   VAR
      sUDT_Status { ExternalAccessible := 'False'; ExternalVisible := 'False'; ExternalWritable := 'False'; S7_SetPoint := 'False'} : "UDT_CommonStatus";   // Common status structure
      sR_TRIG_Automatic {InstructionName := 'R_TRIG'; LibVersion := '1.0'; ExternalAccessible := 'False'; ExternalVisible := 'False'; ExternalWritable := 'False'; S7_SetPoint := 'False'} : R_TRIG;   // Rising edge starting automatic mode
      sR_TRIG_PECOn {InstructionName := 'R_TRIG'; LibVersion := '1.0'; ExternalAccessible := 'False'; ExternalVisible := 'False'; ExternalWritable := 'False'; S7_SetPoint := 'False'} : R_TRIG;   // Rising edge trigger PEC on lift conveyor
      sF_TRIG_TIPLiftConveyor {InstructionName := 'F_TRIG'; LibVersion := '1.0'; ExternalAccessible := 'False'; ExternalVisible := 'False'; ExternalWritable := 'False'; S7_SetPoint := 'False'} : F_TRIG;   // Falling edge trigger TIP signal lift conveyor
      sF_TRIG_PECOff {InstructionName := 'F_TRIG'; LibVersion := '1.0'; ExternalAccessible := 'False'; ExternalVisible := 'False'; ExternalWritable := 'False'; S7_SetPoint := 'False'} : F_TRIG;   // Falling edge trigger PEC on lift conveyor
      sx_AutomaticActive { ExternalAccessible := 'False'; ExternalVisible := 'False'; ExternalWritable := 'False'} : Bool;   // Running in automatic
      sx_LoadIsEmptyTote { ExternalAccessible := 'False'; ExternalVisible := 'False'; ExternalWritable := 'False'} : Bool;   // Load on lift conveyor is an empty tote
      sx_LoadIsFullTote { ExternalAccessible := 'False'; ExternalVisible := 'False'; ExternalWritable := 'False'} : Bool;   // Load on lift conveyor is a full tote
      sx_GetEmptyTote { ExternalAccessible := 'False'; ExternalVisible := 'False'; ExternalWritable := 'False'} : Bool;   // Transport empty tote in
      sx_GetFullTote { ExternalAccessible := 'False'; ExternalVisible := 'False'; ExternalWritable := 'False'} : Bool;   // Transport full tote in
      sx_DeliverEmptyTote { ExternalAccessible := 'False'; ExternalVisible := 'False'; ExternalWritable := 'False'} : Bool;   // Transport empty tote out
      sx_DeliverFullTote { ExternalAccessible := 'False'; ExternalVisible := 'False'; ExternalWritable := 'False'} : Bool;   // Transport full tote out
      sx_EmptyRequest { ExternalAccessible := 'False'; ExternalVisible := 'False'; ExternalWritable := 'False'} : Bool;   // Valid empty request active
      sx_FullRequest { ExternalAccessible := 'False'; ExternalVisible := 'False'; ExternalWritable := 'False'} : Bool;   // Valid full request active
      sx_DoEmptyRequest { ExternalAccessible := 'False'; ExternalVisible := 'False'; ExternalWritable := 'False'} : Bool;   // Handle empty request
      sx_DoFullRequest { ExternalAccessible := 'False'; ExternalVisible := 'False'; ExternalWritable := 'False'} : Bool;   // Handle full request
      sx_Idle { ExternalAccessible := 'False'; ExternalVisible := 'False'; ExternalWritable := 'False'} : Bool;   // Transport is Idle
      si_DistanceToOutfeed { ExternalAccessible := 'False'; ExternalVisible := 'False'; ExternalWritable := 'False'} : Int;   // Actual distance to the end of the lift conveyor
      sx_UpperOutfeedingActive { ExternalAccessible := 'False'; ExternalVisible := 'False'; ExternalWritable := 'False'} : Bool;   // Outfeeding to the upper outfeed is on
      sx_LowerOutfeedingActive { ExternalAccessible := 'False'; ExternalVisible := 'False'; ExternalWritable := 'False'} : Bool;   // Outfeeding to the upper outfeed is on
   END_VAR

   VAR CONSTANT
      ci_Up : Int := 2;
      ci_Down : Int := 1;
      ci_DistanceToOutfeed : Int := 39;   // Distance from middle to the end of the lift conveyor
   END_VAR


BEGIN
	(*
	----------------------------------------------------------------------------------------

	Version
	history:
	Date        | Version   | Author        | Remark
	----------------------------------------------------------------------------------------
	07/04/2023  | 3.0       | F.Baten       | First release TIA 17.5
	14/06/2024  | 3.1       | R.Pieczonka   | Changed handshakes connections, added distance counting while outfeeding

	*)


	REGION 1 - Initial
	    REGION 1.1 - Triggers
	        // Starting automatic
	        #sR_TRIG_Automatic(CLK := #iUDT_VSUInterface.Automatic);

	        // Lift conveyor finished TIP
	        #sF_TRIG_TIPLiftConveyor(CLK := #iqUDT_LiftConveyorHandShake.TIP);

	        // Tote arrived on PEC
	        #sF_TRIG_PECOff(CLK := #ix_PECLift);

	        //Tote gone from PEC
	        #sR_TRIG_PECOn(CLK := #ix_PECLift);

	    END_REGION
	END_REGION

	REGION 7 - Automatic mode

	    REGION 7.1 - Determine load on lift
	        // Lift is in upper position and conveyor is ready to send, the empty tote is loaded on the conveyor.
	        IF #ix_SectionIsUp
	            AND #sx_DoEmptyRequest
	            AND #iUDT_LiftConveyorInterface.VFDRunning
	            AND #sF_TRIG_PECOff.Q
	        THEN
	            #sx_LoadIsEmptyTote := TRUE;
	        END_IF;
	        // Lift is in lower position, and outfeeding empty tote.
	        IF #ix_SectionIsDown
	            AND #iUDT_LiftConveyorInterface.VFDRunning
	            AND #sR_TRIG_PECOn.Q
	            AND #sx_LoadIsEmptyTote
	        THEN
	            #sx_LowerOutfeedingActive := TRUE;
	            #si_DistanceToOutfeed := #ci_DistanceToOutfeed;
	        END_IF;

	        IF #sx_LowerOutfeedingActive
	        THEN
	            #si_DistanceToOutfeed -= #iUDT_LiftConveyorInterface.Displacement;
	        END_IF;
	        //If the ditance from middle conveyor to the end of it is reached,  then the information about tote on the lift is cleared.
	        IF #sx_LowerOutfeedingActive
	            AND #si_DistanceToOutfeed <= 0
	        THEN
	            #sx_LowerOutfeedingActive := FALSE;
	            #sx_LoadIsEmptyTote := FALSE;
	        END_IF;

	        // Lift is in lower position and conveyor is ready to send, the full tote is loaded on the conveyor.
	        IF #ix_SectionIsDown
	            AND #sx_DoFullRequest
	            AND #iUDT_LiftConveyorInterface.VFDRunning
	            AND #sF_TRIG_PECOff.Q
	        THEN
	            #sx_LoadIsFullTote := TRUE;
	        END_IF;
	        // Lift is in upper position, and outfeeding full tote.
	        IF #ix_SectionIsUp
	            AND #iUDT_LiftConveyorInterface.VFDRunning
	            AND #sR_TRIG_PECOn.Q
	            AND #sx_LoadIsFullTote
	        THEN
	            #sx_UpperOutfeedingActive := TRUE;
	            #si_DistanceToOutfeed := #ci_DistanceToOutfeed;
	        END_IF;

	        IF #sx_UpperOutfeedingActive
	        THEN
	            #si_DistanceToOutfeed += #iUDT_LiftConveyorInterface.Displacement;
	        END_IF;
	        //If the ditance from middle conveyor to the end of it is reached, then the information about tote on the lift is cleared.
	        IF #sx_UpperOutfeedingActive
	            AND #si_DistanceToOutfeed <= 0
	        THEN
	            #sx_LoadIsFullTote := FALSE;
	            #sx_UpperOutfeedingActive := FALSE;
	        END_IF;

	        // When starting automatic mode and no load is active but pec still occupied, the load will be set as Full tote.
	        IF NOT #sx_LoadIsFullTote
	            AND NOT #sx_LoadIsEmptyTote
	            AND NOT #ix_PECLift
	            AND #sR_TRIG_Automatic.Q
	        THEN
	            #sx_LoadIsFullTote := TRUE;
	        END_IF;

	        IF #sR_TRIG_Automatic.Q
	        THEN
	            #sx_LowerOutfeedingActive := FALSE;
	            #sx_UpperOutfeedingActive := FALSE;
	        END_IF;
	    END_REGION

	    REGION 7.2 - Request totes
	        // request for empty totes : infeed is full and outfeed is empty and both are automatic active
	        #sx_EmptyRequest := #iqUDT_InfeedEmptyUpHandShake.RTS
	        AND #iqUDT_OutfeedEmptyDownHandShake.RTR
	        AND #ix_ConveyorEmptyInAuto
	        AND #ix_ConveyorEmptyOutAuto;

	        // request for full totes : infeed is full and outfeed is empty and both are automatic active
	        #sx_FullRequest := #iqUDT_InfeedFullDownHandShake.RTS
	        AND #iqUDT_OutfeedFullUpHandshakeUpstream.RTR
	        AND #ix_ConveyorFullInAuto
	        AND #ix_ConveyorFullOutAuto;
	    END_REGION

	    REGION 7.3 - Handle request
	        // Setting reqest to be handled
	        IF #sx_EmptyRequest
	            AND NOT #sx_DoFullRequest
	            AND NOT #sx_LoadIsEmptyTote
	        THEN
	            #sx_DoEmptyRequest := TRUE;
	        ELSIF #sx_FullRequest
	            AND NOT #sx_DoEmptyRequest
	            AND NOT #sx_LoadIsFullTote
	        THEN
	            #sx_DoFullRequest := TRUE;
	        END_IF;

	        // Empty tote is loaded
	        IF (#sx_DoEmptyRequest AND #sx_LoadIsEmptyTote)
	        THEN
	            #sx_DoEmptyRequest := FALSE;
	        END_IF;

	        // Full tote is loaded
	        IF (#sx_DoFullRequest AND #sx_LoadIsFullTote)
	        THEN
	            #sx_DoFullRequest := FALSE;
	        END_IF;

	        // Active request is not valid anymore as lift moved to position
	        IF #sx_DoEmptyRequest AND NOT #sx_EmptyRequest AND #iqUDT_InfeedEmptyUpHandShake.RTS AND #ix_SectionIsUp AND #sx_GetEmptyTote THEN
	            #sx_GetEmptyTote := FALSE;
	            #sx_DoEmptyRequest := FALSE;
	        END_IF;

	        IF #sx_DoFullRequest AND NOT #sx_FullRequest AND #iqUDT_InfeedFullDownHandShake.RTS AND #ix_SectionIsDown AND #sx_GetFullTote THEN
	            #sx_GetFullTote := FALSE;
	            #sx_DoFullRequest := FALSE;
	        END_IF;

	    END_REGION

	    REGION 7.4 - Active Transports
	        // Load empty tote transport is active
	        IF #sx_DoEmptyRequest AND #ix_SectionIsUp
	        THEN
	            #sx_GetEmptyTote := TRUE;
	        END_IF;

	        IF #sx_GetEmptyTote
	            AND
	            ((#iUDT_LiftConveyorInterface.ActualSpeed = 0) AND #sx_LoadIsEmptyTote)
	        THEN
	            #sx_GetEmptyTote := FALSE;
	        END_IF;

	        // Load full tote transport is active
	        IF #sx_DoFullRequest AND #ix_SectionIsDown
	        THEN
	            #sx_GetFullTote := TRUE;
	        END_IF;

	        IF #sx_GetFullTote AND #sx_LoadIsFullTote AND (#iUDT_LiftConveyorInterface.ActualSpeed = 0)
	        THEN
	            #sx_GetFullTote := FALSE;
	        END_IF;

	        // Deliver transports are active
	        #sx_DeliverEmptyTote := #ix_SectionIsDown AND #sx_LoadIsEmptyTote AND (#iUDT_LiftConveyorInterface.ActualSpeed <> 0);
	        #sx_DeliverFullTote := #ix_SectionIsUp AND #sx_LoadIsFullTote AND (#iUDT_LiftConveyorInterface.ActualSpeed <> 0);

	        // Transport is idle
	        #sx_Idle := NOT #sx_GetEmptyTote
	        AND NOT #sx_GetFullTote
	        AND NOT #sx_DeliverFullTote
	        AND NOT #sx_DeliverEmptyTote;
	    END_REGION

	    REGION 7.5 - Lift position request
	        // When lift is at level and transports finished (free to move)
	        // To go to lower level (bring empty tote or get full one)
	        IF #sx_Idle
	            AND ((#ix_SectionIsUp AND #sx_DoFullRequest)
	            OR #sx_LoadIsEmptyTote)
	        THEN
	            #qi_RequestedPosition := #ci_Down;
	        END_IF;

	        // To go to upper level (bring full tote or get empty one)
	        IF #sx_Idle
	            AND ((#ix_SectionIsDown AND #sx_DoEmptyRequest) OR #sx_LoadIsFullTote)
	        THEN
	            #qi_RequestedPosition := #ci_Up;
	        END_IF;

	        #qx_TransportIdle := #sx_Idle;

	    END_REGION

	END_REGION

	REGION 8 - Handshake to conveyors
	    // Reset when not connected
	    #iqUDT_InfeedEmptyUpHandShake.RTR := FALSE;
	    #iqUDT_InfeedFullDownHandShake.RTR := FALSE;

	    #iqUDT_LiftConveyorHandShakeUpstream.GIN := 0;
	    #iqUDT_LiftConveyorHandShakeUpstream.NrOfPosToShift := 0;
	    #iqUDT_OutfeedFullUpHandShake.GIN := 0;
	    #iqUDT_OutfeedFullUpHandShake.NrOfPosToShift := 0;
	    #iqUDT_OutfeedEmptyDownHandShake.GIN := 0;
	    #iqUDT_OutfeedEmptyDownHandShake.NrOfPosToShift := 0;

	    // Direct interface signals when on level
	    IF #ix_SectionIsUp THEN
	        #qx_LiftConveyorDirection := TRUE;                  // Changing direction to left
	        // Infeed
	        #iqUDT_InfeedEmptyUpHandShake.RTR := #iqUDT_LiftConveyorHandShake.RTR AND (#sx_EmptyRequest OR #iqUDT_InfeedEmptyUpHandShake.TIP);
	        #iqUDT_LiftConveyorHandShake.GIN := #iqUDT_InfeedEmptyUpHandShake.GIN;
	        #iqUDT_LiftConveyorHandShakeUpstream.NrOfPosToShift := #iqUDT_InfeedEmptyUpHandShake.NrOfPosToShift;
	        #iqUDT_InfeedEmptyUpHandShake.NrOfPosToShift := 0;
	        #iqUDT_LiftConveyorHandShakeUpstream.RTS := #iqUDT_InfeedEmptyUpHandShake.RTS;
	        //  #iqUDT_HandShakeLiftUp.TIP := #iqUDT_HandShakeEmptyIn.TIP;
	        #iqUDT_LiftConveyorHandShakeUpstream.ResetEnergySave := #iqUDT_InfeedEmptyUpHandShake.ResetEnergySave;

	        // Outfeed
	        #iqUDT_OutfeedFullUpHandshakeUpstream.RTS := #iqUDT_LiftConveyorHandShake.RTS AND #sx_LoadIsFullTote;
	        #iqUDT_OutfeedFullUpHandshakeUpstream.TIP := #iqUDT_LiftConveyorHandShake.TIP;
	        #iqUDT_OutfeedFullUpHandshakeUpstream.GIN := #iqUDT_LiftConveyorHandShake.GIN;
	        #iqUDT_OutfeedFullUpHandshakeUpstream.NrOfPosToShift := #iqUDT_LiftConveyorHandShake.NrOfPosToShift;
	        #iqUDT_LiftConveyorHandShake.NrOfPosToShift := 0;

	        // lift to outfeed transport
	        #iqUDT_LiftConveyorHandShakeUpstream.RTR := #iqUDT_OutfeedFullUpHandshakeUpstream.RTR AND (#sx_LoadIsFullTote OR #iqUDT_LiftConveyorHandShake.TIP);
	    END_IF;

	    IF #ix_SectionIsDown THEN
	        #qx_LiftConveyorDirection := FALSE;                 //Changing direction to right

	        // Infeed Full to lift
	        #iqUDT_InfeedFullDownHandShake.RTR := #iqUDT_LiftConveyorHandShakeUpstream.RTR AND (#sx_FullRequest OR #iqUDT_InfeedFullDownHandShake.TIP);
	        #iqUDT_LiftConveyorHandShakeUpstream.GIN := #iqUDT_InfeedFullDownHandShake.GIN;
	        #iqUDT_LiftConveyorHandShakeUpstream.NrOfPosToShift := #iqUDT_InfeedFullDownHandShake.NrOfPosToShift;
	        #iqUDT_InfeedFullDownHandShake.NrOfPosToShift := 0;
	        #iqUDT_LiftConveyorHandShakeUpstream.RTS := #iqUDT_InfeedFullDownHandShake.RTS;
	        #iqUDT_LiftConveyorHandShakeUpstream.TIP := #iqUDT_InfeedFullDownHandShake.TIP;
	        #iqUDT_LiftConveyorHandShakeUpstream.ResetEnergySave := #iqUDT_InfeedFullDownHandShake.ResetEnergySave;

	        // Outfeed
	        #iqUDT_OutfeedEmptyDownHandshakeUpstream.RTS := #iqUDT_LiftConveyorHandShakeUpstream.RTS AND #sx_LoadIsEmptyTote;
	        #iqUDT_OutfeedEmptyDownHandshakeUpstream.TIP := #iqUDT_LiftConveyorHandShake.TIP;
	        #iqUDT_OutfeedEmptyDownHandshakeUpstream.GIN := #iqUDT_LiftConveyorHandShake.GIN;
	        #iqUDT_OutfeedEmptyDownHandshakeUpstream.NrOfPosToShift := #iqUDT_LiftConveyorHandShake.NrOfPosToShift;
	        #iqUDT_LiftConveyorHandShake.NrOfPosToShift := 0;

	        // lift to outfeed transport
	        #iqUDT_LiftConveyorHandShake.RTR := #iqUDT_OutfeedEmptyDownHandshakeUpstream.RTR AND (#sx_LoadIsEmptyTote OR #iqUDT_LiftConveyorHandShake.TIP);

	    END_IF;

	    #iqUDT_OutfeedFullUpHandshakeUpstream.ResetEnergySave := #iqUDT_InfeedFullDownHandShake.ResetEnergySave
	    OR #iqUDT_LiftConveyorHandShake.ResetEnergySave
	    AND #ix_SectionIsUp;
	    #iqUDT_OutfeedEmptyDownHandshakeUpstream.ResetEnergySave := #iqUDT_InfeedEmptyUpHandShake.ResetEnergySave
	    OR #iqUDT_LiftConveyorHandShake.ResetEnergySave
	    AND #ix_SectionIsDown;

	    //Stop when NOT on level
	    #qx_HoldLiftConveyor := NOT #ix_SectionIsDown AND NOT #ix_SectionIsUp;

	END_REGION

END_FUNCTION_BLOCK

FUNCTION_BLOCK "FB_PECUpdate"
TITLE = FB_PECUpdate
{ S7_Optimized_Access := 'TRUE' }
AUTHOR : MHSE
FAMILY : GeneralSystemFunctions
VERSION : 3.0
// ATTRIBUTES
// AUTO_NUMBER = True
// BLOCK_NUMBER = 221
// END_ATTRIBUTES
//Function block to update parcel data in a tracking array at PEC position.
   VAR_INPUT
      iUDT_PECUpdateConfiguration { ExternalAccessible := 'False'; ExternalVisible := 'False'; ExternalWritable := 'False'} : "UDT_PECUpdateConfiguration";   //   PEC update configuration
      iUDT_ConveyorCommonConfiguration { ExternalAccessible := 'False'; ExternalVisible := 'False'; ExternalWritable := 'False'} : "UDT_ConveyorCommonConfiguration";   //   Conveyor configuration
      ix_PEC { ExternalAccessible := 'False'; ExternalVisible := 'False'; ExternalWritable := 'False'} : Bool;   //   TRUE when the end of section photoeye is not blocked
      ix_TeachingMode { ExternalAccessible := 'False'; ExternalVisible := 'False'; ExternalWritable := 'False'} : Bool;   //   Teaching mode enable
   END_VAR

   VAR_OUTPUT
      qUDT_Status { ExternalAccessible := 'False'; ExternalVisible := 'False'; ExternalWritable := 'False'} : "UDT_PECUpdateStatus";   //   Status structure
      qi_GINwrite { ExternalAccessible := 'False'; ExternalVisible := 'False'; ExternalWritable := 'False'} : Int;   //  Gin found or generated
      qx_PECFiltered { ExternalAccessible := 'False'; ExternalVisible := 'False'; ExternalWritable := 'False'} : Bool;   //   Filtered photoeye signal
   END_VAR

   VAR_IN_OUT
      iqUDT_ConveyorInterface : "UDT_ConveyorInterface";   //   Conveyor interface
      iqUDT_UnknownGINRange : "UDT_UnknownGIN";   //   Unknown GIN
      iqUDT_FifoHeader : "UDT_FifoHeader";   //   FIFO header
      iqUDT_Statistics : "UDT_PECUpdateStatistics";   //   Statistic structure
      iqa_TrackingData : Array[*] of Int;   //   Tracking data
      iqa_FifoData : Array[*] of Int;   //   FIFO data
   END_VAR

   VAR
      sFB_PEC { ExternalAccessible := 'False'; ExternalVisible := 'False'; ExternalWritable := 'False'; S7_SetPoint := 'False'} : "FB_PEC";   //   Photoeye function
      sFB_LengthMeasurement { ExternalAccessible := 'False'; ExternalVisible := 'False'; ExternalWritable := 'False'; S7_SetPoint := 'False'} : "FB_ParcelLength";   //   Length measurement
      sUDT_LostGINFIFOStatus { ExternalAccessible := 'False'; ExternalVisible := 'False'; ExternalWritable := 'False'; S7_SetPoint := 'False'} : "UDT_FifoStatus";   //   Lost GIN FIFO status
      ss_PECDataDeviation { ExternalAccessible := 'False'; ExternalVisible := 'False'; ExternalWritable := 'False'} : Struct   // PEC/Data deviation calculation structure
         Last { ExternalAccessible := 'False'; ExternalVisible := 'False'; ExternalWritable := 'False'} : Int;   //  Last deviation [cm]
         GIN { ExternalAccessible := 'False'; ExternalVisible := 'False'; ExternalWritable := 'False'} : Int;   //  Last GIN deviation
         Sum { ExternalAccessible := 'False'; ExternalVisible := 'False'; ExternalWritable := 'False'} : Int;   //  Deviation sum [cm]
         Nr { ExternalAccessible := 'False'; ExternalVisible := 'False'; ExternalWritable := 'False'} : Int;   //  Deviation number
      END_STRUCT;
      ss_ValidGINRange { ExternalAccessible := 'False'; ExternalVisible := 'False'; ExternalWritable := 'False'} : Struct   //   Valid GIN range
         Start { ExternalAccessible := 'False'; ExternalVisible := 'False'; ExternalWritable := 'False'} : Int;
         End { ExternalAccessible := 'False'; ExternalVisible := 'False'; ExternalWritable := 'False'} : Int;
         GIN { ExternalAccessible := 'False'; ExternalVisible := 'False'; ExternalWritable := 'False'} : Int;
      END_STRUCT;
      ss_AlignedParcelsCounters { ExternalAccessible := 'False'; ExternalVisible := 'False'; ExternalWritable := 'False'} : Struct   //   Aligned parcels counters
         Total { ExternalAccessible := 'False'; ExternalVisible := 'False'; ExternalWritable := 'False'} : Int;   //   Total aligned parcels
         DataNoPEC { ExternalAccessible := 'False'; ExternalVisible := 'False'; ExternalWritable := 'False'} : Int;   //   Parcels aligned in case data detected without photoeye signal
         PECNoData { ExternalAccessible := 'False'; ExternalVisible := 'False'; ExternalWritable := 'False'} : Int;   //   Parcels aligned in case parcel detected without data
      END_STRUCT;
      ss_LostParcelsCounters { ExternalAccessible := 'False'; ExternalVisible := 'False'; ExternalWritable := 'False'} : Struct   //   Lost parcels counters
         Total { ExternalAccessible := 'False'; ExternalVisible := 'False'; ExternalWritable := 'False'} : Int;   //   Total number of lost parcels
         DoubleData { ExternalAccessible := 'False'; ExternalVisible := 'False'; ExternalWritable := 'False'} : Int;   //   Parcels lost due to double data found in a search window
         ParcelNotFound { ExternalAccessible := 'False'; ExternalVisible := 'False'; ExternalWritable := 'False'} : Int;   //   Parcels lost due to no parcel detected after travelling search window distance
      END_STRUCT;
      ss_LostValidParcelsCounters { ExternalAccessible := 'False'; ExternalVisible := 'False'; ExternalWritable := 'False'} : Struct   //   Lost parcels counters
         Total { ExternalAccessible := 'False'; ExternalVisible := 'False'; ExternalWritable := 'False'} : Int;   //   Total number of lost parcels
         DoubleData { ExternalAccessible := 'False'; ExternalVisible := 'False'; ExternalWritable := 'False'} : Int;   //   Parcels lost due to double data found in a search window
         ParcelNotFound { ExternalAccessible := 'False'; ExternalVisible := 'False'; ExternalWritable := 'False'} : Int;   //   Parcels lost due to no parcel detected after travelling search window distance
      END_STRUCT;
      si_UnknownParcelsCounters { ExternalAccessible := 'False'; ExternalVisible := 'False'; ExternalWritable := 'False'} : Struct   //   Unknown parcels counters
         Total { ExternalAccessible := 'False'; ExternalVisible := 'False'; ExternalWritable := 'False'} : Int;   //   Total number of unknown parcels
         LostParcelFound { ExternalAccessible := 'False'; ExternalVisible := 'False'; ExternalWritable := 'False'} : Int;   //   Parcel found with a lost data, unknown GIN created
         DataNotFound { ExternalAccessible := 'False'; ExternalVisible := 'False'; ExternalWritable := 'False'} : Int;   //   Data not found during search window scan
      END_STRUCT;
      sR_TRIG_Parcel {InstructionName := 'R_TRIG'; LibVersion := '1.0'; ExternalAccessible := 'False'; ExternalVisible := 'False'; ExternalWritable := 'False'; S7_SetPoint := 'False'} : R_TRIG;   //   Parcel detected rising edge to count parcels
      sR_TRIG_ParcelFound {InstructionName := 'R_TRIG'; LibVersion := '1.0'; ExternalAccessible := 'False'; ExternalVisible := 'False'; ExternalWritable := 'False'; S7_SetPoint := 'False'} : R_TRIG;   //   Parcel detected rising edge to update the PEC position tracking record
      sR_TRIG_DataFound {InstructionName := 'R_TRIG'; LibVersion := '1.0'; ExternalAccessible := 'False'; ExternalVisible := 'False'; ExternalWritable := 'False'; S7_SetPoint := 'False'} : R_TRIG;   //   Any data found at a PEC position rising edge
      sR_TRIG_PositiveDataFound {InstructionName := 'R_TRIG'; LibVersion := '1.0'; ExternalAccessible := 'False'; ExternalVisible := 'False'; ExternalWritable := 'False'; S7_SetPoint := 'False'} : R_TRIG;   //   Positive data found at a PEC position rising edge
      sR_TRIG_TeachMode {InstructionName := 'R_TRIG'; LibVersion := '1.0'; ExternalAccessible := 'False'; ExternalVisible := 'False'; ExternalWritable := 'False'; S7_SetPoint := 'False'} : R_TRIG;   //   Teaching mode activation rising edge
      sR_TRIG_TooManyLost {InstructionName := 'R_TRIG'; LibVersion := '1.0'; ExternalAccessible := 'False'; ExternalVisible := 'False'; ExternalWritable := 'False'; S7_SetPoint := 'False'} : R_TRIG;   //   Too many lost parcels error statistics trigger
      slr_Performance { ExternalAccessible := 'False'; ExternalVisible := 'False'; ExternalWritable := 'False'} : LReal := 100.0;   //   Update performance [%]
      sdi_TotalNumberOfParcels { ExternalAccessible := 'False'; ExternalVisible := 'False'; ExternalWritable := 'False'} : DInt;   //   Total number of parcels detected
      sdi_TotalNumberOfData { ExternalAccessible := 'False'; ExternalVisible := 'False'; ExternalWritable := 'False'} : DInt;   //   Total number of data detected
      si_PECPosition { ExternalAccessible := 'False'; ExternalVisible := 'False'; ExternalWritable := 'False'} : Int;   //   Photoeye position [cm]
      si_SearchWindow { ExternalAccessible := 'False'; ExternalVisible := 'False'; ExternalWritable := 'False'} : Int;   //   Data search distance from photoeye position [cm]
      si_GINToWrite { ExternalAccessible := 'False'; ExternalVisible := 'False'; ExternalWritable := 'False'} : Int;   //   Found or generated GIN, which will be used to update photoeye position in the tracking array
      si_PositionToUpdate { ExternalAccessible := 'False'; ExternalVisible := 'False'; ExternalWritable := 'False'} : Int;   //   Position in a tracking array to be updated
      si_Direction { ExternalAccessible := 'False'; ExternalVisible := 'False'; ExternalWritable := 'False'} : Int;   //   Direction of the displacement to parametrize loops
      si_Displacement { ExternalAccessible := 'False'; ExternalVisible := 'False'; ExternalWritable := 'False'} : Int;   //   Displacement [cm]
      si_ParcelWaitDistance { ExternalAccessible := 'False'; ExternalVisible := 'False'; ExternalWritable := 'False'} : Int;   //   Parcel delay [cm]
      si_LastUpdatedGIN { ExternalAccessible := 'False'; ExternalVisible := 'False'; ExternalWritable := 'False'} : Int;   //   Last updated GIN to check if next data is a new one
      si_LastCountedData { ExternalAccessible := 'False'; ExternalVisible := 'False'; ExternalWritable := 'False'} : Int;   //   Last counted data
      si_LostParcelsInARow { ExternalAccessible := 'False'; ExternalVisible := 'False'; ExternalWritable := 'False'} : Int;   //   Number of lost parcel in a row
      si_NumberOfTeachedParcels { ExternalAccessible := 'False'; ExternalVisible := 'False'; ExternalWritable := 'False'} : Int;   //   Number of teached parcels
      si_AverageSlip { ExternalAccessible := 'False'; ExternalVisible := 'False'; ExternalWritable := 'False'} : Int;   //   Average parcel slip [cm]
      si_CalculatedLengthCorrection { ExternalAccessible := 'False'; ExternalVisible := 'False'; ExternalWritable := 'False'} : Int;   //   Calculated length correction after teaching
      si_ParcelLengthFilterCounter { ExternalAccessible := 'False'; ExternalVisible := 'False'; ExternalWritable := 'False'} : Int;   //  Parcel length filter counter [cm]
      si_ParcelLengthFilterOldGIN { ExternalAccessible := 'False'; ExternalVisible := 'False'; ExternalWritable := 'False'} : Int;   //  Parcel length filter old GIN
      si_LoopCounter { ExternalAccessible := 'False'; ExternalVisible := 'False'; ExternalWritable := 'False'} : Int;   //   Loop counter
      sx_ParcelDetected { ExternalAccessible := 'False'; ExternalVisible := 'False'; ExternalWritable := 'False'} : Bool;   //   Parcel detected
      sx_ParcelWaitEnable { ExternalAccessible := 'False'; ExternalVisible := 'False'; ExternalWritable := 'False'} : Bool;   //   Missing parcel monitoring
      sx_TeachingMode { ExternalAccessible := 'False'; ExternalVisible := 'False'; ExternalWritable := 'False'} : Bool;   //   Teaching mode
      sx_GenerateGIN { ExternalAccessible := 'False'; ExternalVisible := 'False'; ExternalWritable := 'False'} : Bool;   //   Request to generate GIN
      sx_LostGINFIFOError { ExternalAccessible := 'False'; ExternalVisible := 'False'; ExternalWritable := 'False'} : Bool;   //   Lost GIN FIFO error
      sx_LostGINFIFOWarning { ExternalAccessible := 'False'; ExternalVisible := 'False'; ExternalWritable := 'False'} : Bool;   //   Lost GIN FIFO warning
      sx_InvalidDirection { ExternalAccessible := 'False'; ExternalVisible := 'False'; ExternalWritable := 'False'} : Bool;   //   Invalid direction
      sx_InvalidGINRange { ExternalAccessible := 'False'; ExternalVisible := 'False'; ExternalWritable := 'False'} : Bool;   //   Invalid GIN range
      sx_InvalidDisplacement { ExternalAccessible := 'False'; ExternalVisible := 'False'; ExternalWritable := 'False'} : Bool;   //   Invalid displacement
      sx_InvalidSearchWindow { ExternalAccessible := 'False'; ExternalVisible := 'False'; ExternalWritable := 'False'} : Bool;   //   Invalid search window
      sx_DoubleDataFound { ExternalAccessible := 'False'; ExternalVisible := 'False'; ExternalWritable := 'False'} : Bool;   //   Double data detected
      sx_LengthMeasurementEnable { ExternalAccessible := 'False'; ExternalVisible := 'False'; ExternalWritable := 'False'} : Bool;
   END_VAR

   VAR_TEMP
      tUDT_PECConfiguration : "UDT_PECConfiguration";   //   PEC configuration
      tUDT_PECStatus : "UDT_PECStatus";   //   PEC status
   END_VAR

   VAR CONSTANT
      ci_ZeroGIN : Int;   //   GIN = 0
   END_VAR


BEGIN
	(*
	----------------------------------------------------------------------------------------

	Version history:
	Date        | Version   | Author        | Remark
	----------------------------------------------------------------------------------------
	24/05/2019  | 0.1       | L.Klar        | first release MHSE TIA 15.1
	13/06/2019  | 0.2       | A.Nowak       | Replacement of instruction if for direct write into variable
	21/06/2019  | 0.3       | A.Nowak       | Add gap mesurement function and reorganise block (regions)
	24/07/2019  | 2.0       | L.Klar        | 2.0 MHSE library release TIA 15.1
	23/08/2019  | 2.1       | L.Klar        | "UDT_ConveyorConfiguration" changed to "UDT_ConveyorCommonConfiguration"
	XX/08/2019  | 2.2       | L.Klar        | Update logic changed
	19/09/2019  | 2.3       | P.Majka       | Updating checking PEC and PEC filtered signals
	30/09/2019  | 2.4       | L.Klar        | FB_PEC added, Filtered PEC signal output added
	21/10/2019  | 2.6       | L.Klar        | Configuration UDT chanaged to input, PEC configuration interface input name changed
	23/10/2019  | 2.7       | P.Majka       | Added Region 1, renumerating Regions, changed logic in Region 10.3 and Region 5
	29/10/2019  | 2.8       | L.Klar        | FB_PEC call changed
	14/11/2019  | 2.9       | L.Klar        | Deviations calculation corrected
	14/11/2019  | 3.0       | P.Majka       | 3.0 MHSE library release TIA 15.1
	20/12/2019  | 3.1       | S.Deulkar     | Used configureation error bit to report to conveyor block
	07/01/2020  | 3.2       | L.Klar        | GIN record structure updated, GIN cleared with default one during generation
	                                        | PECUpdate configuration UDT update - search window DINT -> INT,
	                                        | Conveyor common configuration UDT update - length INT -> DINT  conversion added
	29/01/2020  | 3.3       | L.Klar        | Negative GIN handling fixed, configuration bit added to delete negative GIN instead of ignoing it.
	24/02/2020  | 3.4       | L.Klar        | Formating changes, statistics counter added
	10/03/2020  | 3.5       | F.Baten       | Range check unknown GIN region 7
	26/03/2020  | 3.6       | F.Baten       | Added output 'qi_GINwrite'
	25/11/2020  | 3.7       | L.Klar        | Length filter added
	07/12/2020  | 3.8       | L.Klar        | Length filter bug fix
	22/01/2021  | 3.9       | L.Klar        | Total number of parcels and lost parcels counter fixed
	14/08/2021  | 3.10      | S. Deulkar    | Update from EMA
	21/02/2023  | 4.0       | F.Baten       | 4.0 Release TIA 17.5
	*)


	REGION 1 – FIFO header status update

	    "FC_Fifo"(ic_Mode := 'S',
	              qUDT_Status => #sUDT_LostGINFIFOStatus,
	              qx_Error => #sx_LostGINFIFOError,
	              qx_Warning => #sx_LostGINFIFOWarning,
	              iqv_Data := #si_GINToWrite,
	              iqUDT_FifoHeader := #iqUDT_FifoHeader,
	              iqv_DataBuffer := #iqa_FifoData);

	END_REGION

	REGION 2 – Displacement read

	    #si_Displacement := #iqUDT_ConveyorInterface.Displacement;

	END_REGION

	REGION 3 – PEC Position conversion from mm to cm

	    // The conversion is required because the photoeye position is given in mm and the tracking resolution is 1 cm.
	    #si_PECPosition := DINT_TO_INT(#iUDT_PECUpdateConfiguration.Distance / 10);

	END_REGION

	REGION 4 – Teaching mode enable

	    (* Teaching mode is used to calculate conveyor length correction, which allows to align real conveyor length with a tracking array length.
	       Correction is calculated as a difference between photoeye signal and tracking data deviations.
	       Calculated correction has to be manually copied from a FB_PECUpdate instance data block to conveyor configuration.*)

	    // Teaching mode is initialized and activated manually via block input.
	    #sR_TRIG_TeachMode(CLK := #ix_TeachingMode);

	    IF (#sR_TRIG_TeachMode.Q
	        AND NOT #sx_TeachingMode)
	    THEN
	        #ss_PECDataDeviation.Nr := 0;
	        #ss_PECDataDeviation.Sum := 0;
	        #si_NumberOfTeachedParcels := 0;
	        #sx_TeachingMode := TRUE;
	    END_IF;

	END_REGION

	REGION 5 – Photoeye

	    (*FB_PEC block call to filter photoeye signal and calculate jam status.*)

	    // Copy PEC configuration.
	    #tUDT_PECConfiguration.Distance := #iUDT_PECUpdateConfiguration.Distance;
	    #tUDT_PECConfiguration.JamDisplacementLimit := #iUDT_PECUpdateConfiguration.JamDisplacementLimit;
	    #tUDT_PECConfiguration.TimeOnDelay := #iUDT_PECUpdateConfiguration.TimeOnDelay;
	    #tUDT_PECConfiguration.TimeOffDelay := #iUDT_PECUpdateConfiguration.TimeOffDelay;
	    #tUDT_PECConfiguration.ResetWithPECBlocked := #iUDT_PECUpdateConfiguration.ResetWithPECBlocked;

	    //Call FB_PEC.
	    #sFB_PEC(ix_PEC := #ix_PEC,
	             iUDT_PECConfiguration := #tUDT_PECConfiguration,
	             qUDT_HMIStatus => #tUDT_PECStatus,
	             iqUDT_ConveyorInterface := #iqUDT_ConveyorInterface,
	             iqUDT_PECStatistics := #iqUDT_Statistics.PEC);

	    // Parcel length filter
	    IF NOT #ix_PEC
	        AND #iUDT_PECUpdateConfiguration.ParcelLengthFilter
	        AND #iqa_TrackingData[#si_PECPosition - 1] > 0
	        AND #iqa_TrackingData[#si_PECPosition - 1] <> #si_ParcelLengthFilterOldGIN THEN

	        IF "DB_GIN".GIN[#iqa_TrackingData[#si_PECPosition - 1]].General.Length > 0 THEN
	            #si_ParcelLengthFilterCounter := "DB_GIN".GIN[#iqa_TrackingData[#si_PECPosition - 1]].General.Length;
	        END_IF;

	        #si_ParcelLengthFilterOldGIN := #iqa_TrackingData[#si_PECPosition - 1];

	    END_IF;

	    IF #si_ParcelLengthFilterCounter > 0 THEN

	        #qUDT_Status.PEC := FALSE;
	        #qx_PECFiltered := FALSE;
	        #si_ParcelLengthFilterCounter -= #iqUDT_ConveyorInterface.Displacement;

	    ELSE

	        #qUDT_Status.PEC := #sFB_PEC.qx_PECFiltered;
	        #qx_PECFiltered := #sFB_PEC.qx_PECFiltered;

	    END_IF;

	    #qUDT_Status.Jam := #tUDT_PECStatus.Jam;

	    // Parcel detected variable to simplify further photoeye position tracking record update.
	    #sx_ParcelDetected := NOT #qUDT_Status.PEC;

	END_REGION

	REGION 6 – Error reset

	    // Reset errors when reset signal is given.
	    IF (#iqUDT_ConveyorInterface.InternalErrorReset)
	    THEN
	        #si_LostParcelsInARow := 0;
	        #qUDT_Status.TooManyLost := FALSE;
	        #sx_InvalidDisplacement := FALSE;
	    END_IF;

	END_REGION

	REGION 7 – GIN generator initialization

	    // Valid GIN range configuration is moved to a structure.
	    #ss_ValidGINRange.Start := #iUDT_PECUpdateConfiguration.GINRangeStart;
	    #ss_ValidGINRange.End := #iUDT_PECUpdateConfiguration.GINRangeEnd;

	    // Check if the unknown GIN is within range
	    IF #iqUDT_UnknownGINRange.GIN < #iqUDT_UnknownGINRange.Start
	        OR #iqUDT_UnknownGINRange.GIN > #iqUDT_UnknownGINRange.End
	    THEN
	        #iqUDT_UnknownGINRange.GIN := #iqUDT_UnknownGINRange.Start;
	    END_IF;

	    // Whenever valid GIN range is changed and the generated GIN doesn't fit, it's initialized.
	    IF (#ss_ValidGINRange.GIN < #ss_ValidGINRange.Start
	        OR #ss_ValidGINRange.GIN > #ss_ValidGINRange.End)
	    THEN
	        #ss_ValidGINRange.GIN := #ss_ValidGINRange.Start;
	    END_IF;

	    // Valid GIN range is set locally in PEC update configuration structure and it can't overlap with a global unknown GIN range.
	    #sx_InvalidGINRange := #iUDT_PECUpdateConfiguration.GenerationPoint
	    AND (#ss_ValidGINRange.End <= #ss_ValidGINRange.Start
	    OR #ss_ValidGINRange.Start <= #iqUDT_UnknownGINRange.End
	    OR #iqUDT_UnknownGINRange.End <= #iqUDT_UnknownGINRange.Start)
	    AND #ss_ValidGINRange.Start < 1000;   // Until 1000 it is UFO range

	END_REGION

	REGION 8 – Search window and displacement validation

	    (*Both parameters have to be checked to prevent tracking array exceeding.*)

	    // Search window cannot be lower than zero and greater than distance between PEC position and conveyor edge.
	    #sx_InvalidSearchWindow := #iUDT_PECUpdateConfiguration.SearchWindowFwd < 0
	    OR #iUDT_PECUpdateConfiguration.SearchWindowFwd >= #iUDT_ConveyorCommonConfiguration.Length + #iUDT_ConveyorCommonConfiguration.LengthCorrection - #si_PECPosition
	    OR #iUDT_PECUpdateConfiguration.SearchWindowRvs < 0
	    OR #iUDT_PECUpdateConfiguration.SearchWindowRvs >= #si_PECPosition;

	    // Displacement cannot be greater than the photoeye position.
	    IF (ABS(#si_Displacement) > #si_PECPosition)
	    THEN
	        #sx_InvalidDisplacement := TRUE;
	    END_IF;

	END_REGION

	REGION 9 – Total number of parcels counter

	    (*Parcels are counted basing on parcel detection rising edge trigger. Counting is blocked
	      during PLC first scan, when photoeye signal becomes 0.*)

	    #sR_TRIG_Parcel(CLK := #sx_ParcelDetected);

	    IF (#sR_TRIG_Parcel.Q
	        AND NOT "DB_Memory".FirstScan)
	    THEN
	        // Total number of parcels.
	        #sdi_TotalNumberOfParcels += 1;

	        // Every detected parcel resets lost parcels in a row counter.
	        #si_LostParcelsInARow := 0;

	        // Number of teached parcels is incremented if teaching mode is activated.
	        IF (#sx_TeachingMode)
	        THEN
	            #si_NumberOfTeachedParcels += 1;
	        END_IF;
	    END_IF;

	END_REGION

	REGION 10 – PEC Update
	    (* Photoeye position record is updated after every tracking register shift, basing on
	       actual situation - photoeye signal and data availability. In case of displacement
	       graeter than one, the loop will be executed the proper number of times. The update loop
	       can be executed if there is no configuration errors and the displacement was given.*)

	    WHILE #si_Displacement <> 0
	        AND NOT #sx_InvalidGINRange
	        AND NOT #sx_InvalidDisplacement
	        AND NOT #sx_InvalidSearchWindow
	    DO

	        REGION 10.1 – Direction

	            (*Depending on displacement sign, the direction of movement is determinated. This allows to choose
	            ` correct search window and parametrize all search loops to count up or down.*)

	            IF (#si_Displacement < 0)
	            THEN
	                #si_Direction := -1;
	                #si_SearchWindow := #iUDT_PECUpdateConfiguration.SearchWindowRvs;
	            ELSIF (#si_Displacement > 0)
	            THEN
	                #si_Direction := 1;
	                #si_SearchWindow := #iUDT_PECUpdateConfiguration.SearchWindowFwd;
	            END_IF;

	        END_REGION

	        REGION 10.2 – Position to update

	            // Position pointer used to specify the tracking array record to be updated.
	            #si_PositionToUpdate := #si_PECPosition - #si_Displacement + #si_Direction;

	        END_REGION


	        REGION 10.3 – Total number of data counter

	            (*Total number of data is incremented every time when new GIN is detected.*)

	            IF (#iqa_TrackingData[#si_PositionToUpdate + 1] > 0
	                AND #iqa_TrackingData[#si_PositionToUpdate + 1] <> #si_LastCountedData)
	            THEN
	                #sdi_TotalNumberOfData += 1;
	                #si_LastCountedData := #iqa_TrackingData[#si_PositionToUpdate + 1];
	            END_IF;

	        END_REGION

	        REGION 10.4 – GIN detection

	            (* Data found and parcel found triggers are used to determine the update case,
	               whether the data occurred first or a parcel.*)

	            // Trigger on any data found at a PEC position to detect the front of the parcel data.
	            #sR_TRIG_DataFound(CLK := #iqa_TrackingData[#si_PositionToUpdate] <> 0);

	            // Trigger on positive data found at a PEC position to detect the front of the parcel data.
	            #sR_TRIG_PositiveDataFound(CLK := #iqa_TrackingData[#si_PositionToUpdate] > 0);

	            // Trigger to detect front of the parcel.
	            #sR_TRIG_ParcelFound(CLK := #sx_ParcelDetected);

	(*
	Data detected without PEC signal

	                         Search window
	                          <--------|
	Data                              PEC
	|----------------------------------|------------------------------------------|
	|                           XXXXXXXX                                          |
	|----------------------------------|------------------------------------------|
	                                   |
	Conveyor                           |
	|----------------------------------|------------------------------------------|
	|                      YYYYYYYY    |                                          |
	|                      YYYYYYYY    |                                          |
	|                      YYYYYYYY    |                                          |
	|----------------------------------|------------------------------------------|
	*)
	(* Data detected without PEC signal.*)
	            IF (#sR_TRIG_PositiveDataFound.Q
	                AND NOT #sx_ParcelDetected)
	            THEN
	                #si_GINToWrite := 0;
	                // Double data detection loop.
	                FOR #si_LoopCounter := #si_PositionToUpdate TO
	                    #si_PECPosition + (#si_SearchWindow * #si_Direction) BY #si_Direction DO
	                    // Data found in a search window.
	                    IF (#iqa_TrackingData[#si_LoopCounter] > 0)
	                    THEN
	                        // First GIN found.
	                        IF (#si_GINToWrite = 0)
	                        THEN
	                            // Get the GIN if it's different than last updated GIN.
	                            IF #iqa_TrackingData[#si_LoopCounter] <> #si_LastUpdatedGIN THEN
	                                #si_GINToWrite := #iqa_TrackingData[#si_LoopCounter];
	                            END_IF;
	                            // If the first GIN was found, the scan loop conitues to check if there is no other data.
	                        ELSE
	                            // Next found data is different than the first one. Double data detected.
	                            IF (#iqa_TrackingData[#si_LoopCounter] <> #si_GINToWrite)
	                            THEN
	                                #sx_DoubleDataFound := TRUE;
	                                // First found GIN is marked as a lost one and the GIN is stored in a FIFO register.
	                                IF ("DB_GIN".GIN[#si_GINToWrite].General.Lost = FALSE)
	                                THEN
	                                    "DB_GIN".GIN[#si_GINToWrite].General.Lost := TRUE;

	                                    "FC_Fifo"(ic_Mode := 'W',
	                                              qUDT_Status => #sUDT_LostGINFIFOStatus,
	                                              qx_Error => #sx_LostGINFIFOError,
	                                              qx_Warning => #sx_LostGINFIFOWarning,
	                                              iqv_Data := #si_GINToWrite,
	                                              iqUDT_FifoHeader := #iqUDT_FifoHeader,
	                                              iqv_DataBuffer := #iqa_FifoData);

	                                    // Update statistics
	                                    #ss_LostParcelsCounters.Total += 1;
	                                    #ss_LostParcelsCounters.DoubleData += 1;


	                                    ////////////////////

	                                    IF #si_GINToWrite >= 1000 THEN
	                                        #ss_LostValidParcelsCounters.Total += 1;
	                                        #ss_LostValidParcelsCounters.DoubleData += 1;
	                                    END_IF;

	                                    ////////////////
	                                END_IF;

	                                // Second found GIN is marked as a lost one and the GIN is stored in a FIFO register.
	                                IF ("DB_GIN".GIN[#iqa_TrackingData[#si_LoopCounter]].General.Lost = FALSE)
	                                THEN
	                                    "DB_GIN".GIN[#iqa_TrackingData[#si_LoopCounter]].General.Lost := TRUE;

	                                    "FC_Fifo"(ic_Mode := 'W',
	                                              qUDT_Status => #sUDT_LostGINFIFOStatus,
	                                              qx_Error => #sx_LostGINFIFOError,
	                                              qx_Warning => #sx_LostGINFIFOWarning,
	                                              iqv_Data := #iqa_TrackingData[#si_LoopCounter],
	                                              iqUDT_FifoHeader := #iqUDT_FifoHeader,
	                                              iqv_DataBuffer := #iqa_FifoData);

	                                    // Update statistics
	                                    #ss_LostParcelsCounters.Total += 1;
	                                    #ss_LostParcelsCounters.DoubleData += 1;

	                                    ////////////////////

	                                    IF #iqa_TrackingData[#si_LoopCounter] >= 1000 THEN
	                                        #ss_LostValidParcelsCounters.Total += 1;
	                                        #ss_LostValidParcelsCounters.DoubleData += 1;
	                                    END_IF;

	                                    ////////////////
	                                    //
	                                END_IF;
	                                // Stop search window scan in case of double data detection
	                                EXIT;
	                            END_IF;
	                        END_IF;
	                    END_IF;
	                END_FOR;

	                // Becasue the data was found as a first one, GIN is stored and the logic to wait for a parcel is enebaled.
	                // If the double data was found there is no need to wait for a parcel. Data has been marked as a lost one.
	                IF NOT #sx_DoubleDataFound
	                THEN
	                    #sx_ParcelWaitEnable := TRUE;
	                END_IF;

	                #sx_DoubleDataFound := FALSE;
	(*
	Data and PEC signal detected at the same time - perfect match

	                         Search window
	                          <--------|
	Data                              PEC
	|----------------------------------|------------------------------------------|
	|                           XXXXXXXX                                          |
	|----------------------------------|------------------------------------------|
	                                   |
	Conveyor                           |
	|----------------------------------|------------------------------------------|
	|                           XXXXXXXX                                          |
	|                           XXXXXXXX                                          |
	|                           XXXXXXXX                                          |
	|----------------------------------|------------------------------------------|

	or PEC signal found without data or with old ones

	                         Search window
	                          <--------|
	Data                              PEC
	|----------------------------------|------------------------------------------|
	|                    XXXXXXXX      |                                          |
	|----------------------------------|------------------------------------------|
	                                   |
	Conveyor                           |
	|----------------------------------|------------------------------------------|
	|                           XXXXXXXX                                          |
	|                           XXXXXXXX                                          |
	|                           XXXXXXXX                                          |
	|----------------------------------|------------------------------------------|
	*)
	(*Data and PEC signal detected at the same time (perfect match) or PEC signal found without data or with old ones.*)
	            ELSIF (#sR_TRIG_ParcelFound.Q
	                AND (#sR_TRIG_PositiveDataFound.Q
	                OR (#iqa_TrackingData[#si_PositionToUpdate] = 0
	                OR #iqa_TrackingData[#si_PositionToUpdate] = #si_LastUpdatedGIN)
	                AND NOT #sx_ParcelWaitEnable))
	            THEN
	                // If the PEC is set as a GIN generation point, skip data detection loop and go to GIN generator.
	                IF (#iUDT_PECUpdateConfiguration.GenerationPoint)
	                THEN
	                    #sx_GenerateGIN := TRUE;
	                    // If the the PEC isn't a generation point, data search loop is enabled.
	                ELSE
	                    #si_GINToWrite := 0;

	                    // Double data detection loop.
	                    FOR #si_LoopCounter := #si_PositionToUpdate TO
	                        #si_PECPosition + (#si_SearchWindow * #si_Direction) BY #si_Direction DO

	                        // Data found in a search window.
	                        IF (#iqa_TrackingData[#si_LoopCounter] > 0)
	                        THEN
	                            // First GIN found.
	                            IF (#si_GINToWrite = 0)
	                            THEN
	                                // Get the GIN if it's different than last updated GIN.
	                                IF #iqa_TrackingData[#si_LoopCounter] <> #si_LastUpdatedGIN THEN
	                                    #si_GINToWrite := #iqa_TrackingData[#si_LoopCounter];

	                                    // PEC/Data deviation acquisition
	                                    #ss_PECDataDeviation.Last := DINT_TO_INT(#si_PECPosition - #si_LoopCounter);
	                                    #ss_PECDataDeviation.GIN := #si_GINToWrite;
	                                    #ss_PECDataDeviation.Sum -= ABS(#ss_PECDataDeviation.Last);
	                                    #ss_PECDataDeviation.Nr += 1;

	                                    // Parcel aligned statistics
	                                    IF (ABS(#ss_PECDataDeviation.Last) > ABS(#si_Displacement - 1))
	                                    THEN
	                                        #ss_AlignedParcelsCounters.Total += 1;
	                                        #ss_AlignedParcelsCounters.PECNoData += 1;
	                                    END_IF;
	                                END_IF;
	                                // If the first GIN was found, the scan loop conitues to check if there is no other data.
	                            ELSE
	                                // Next found data is different than the first one. Double data detected.
	                                IF (#iqa_TrackingData[#si_LoopCounter] <> #si_GINToWrite)
	                                THEN
	                                    // First found GIN is marked as a lost one and the GIN is stored in a FIFO register.
	                                    IF ("DB_GIN".GIN[#si_GINToWrite].General.Lost = FALSE)
	                                    THEN
	                                        "DB_GIN".GIN[#si_GINToWrite].General.Lost := TRUE;
	                                        "FC_Fifo"(ic_Mode := 'W',
	                                                  qUDT_Status => #sUDT_LostGINFIFOStatus,
	                                                  qx_Error => #sx_LostGINFIFOError,
	                                                  qx_Warning => #sx_LostGINFIFOWarning,
	                                                  iqv_Data := #si_GINToWrite,
	                                                  iqUDT_FifoHeader := #iqUDT_FifoHeader,
	                                                  iqv_DataBuffer := #iqa_FifoData);

	                                        // Update statistics
	                                        #ss_LostParcelsCounters.Total += 1;
	                                        #ss_LostParcelsCounters.DoubleData += 1;

	                                        ////////////////////

	                                        IF #si_GINToWrite >= 1000 THEN
	                                            #ss_LostValidParcelsCounters.Total += 1;
	                                            #ss_LostValidParcelsCounters.DoubleData += 1;
	                                        END_IF;

	                                        ////////////////
	                                        //
	                                    END_IF;

	                                    // Second found GIN is marked as a lost one and the GIN is stored in a FIFO register.
	                                    IF ("DB_GIN".GIN[#iqa_TrackingData[#si_LoopCounter]].General.Lost = FALSE)
	                                    THEN
	                                        "DB_GIN".GIN[#iqa_TrackingData[#si_LoopCounter]].General.Lost := TRUE;
	                                        "FC_Fifo"(ic_Mode := 'W',
	                                                  qUDT_Status => #sUDT_LostGINFIFOStatus,
	                                                  qx_Error => #sx_LostGINFIFOError,
	                                                  qx_Warning => #sx_LostGINFIFOWarning,
	                                                  iqv_Data := #iqa_TrackingData[#si_LoopCounter],
	                                                  iqUDT_FifoHeader := #iqUDT_FifoHeader,
	                                                  iqv_DataBuffer := #iqa_FifoData);

	                                        // Update statistics
	                                        #ss_LostParcelsCounters.Total += 1;
	                                        #ss_LostParcelsCounters.DoubleData += 1;

	                                        ////////////////////

	                                        IF #iqa_TrackingData[#si_LoopCounter] >= 1000 THEN
	                                            #ss_LostValidParcelsCounters.Total += 1;
	                                            #ss_LostValidParcelsCounters.DoubleData += 1;
	                                        END_IF;

	                                        ////////////////
	                                        //
	                                    END_IF;
	                                    // Stop search window scan in case of double data detection
	                                    EXIT;
	                                END_IF;
	                            END_IF;
	                        END_IF;
	                    END_FOR;

	                    // GIN not found in a search window
	                    IF (#si_GINToWrite = 0)
	                    THEN
	                        #sx_GenerateGIN := TRUE;
	                        #si_UnknownParcelsCounters.DataNotFound += 1;
	                    END_IF;

	                    // Found GIN is a lost one - generate unknown GIN
	                    // Found GIN isn't lost or it's negative - don't do anything
	                    IF (#si_GINToWrite > 0)
	                    THEN
	                        IF ("DB_GIN".GIN[#si_GINToWrite].General.Lost)
	                        THEN
	                            #sx_GenerateGIN := TRUE;
	                            #si_UnknownParcelsCounters.LostParcelFound += 1;
	                        END_IF;
	                    END_IF;
	                END_IF;

	                (*Second parcel has been found during data update. Situation can occur when search window is too short
	                  and the data is shifted. In that case found GIN will be marked as a lost one and new unknown GIN will be
	                  generated. Negative GIN will be ignored.*)
	            ELSIF (#sR_TRIG_ParcelFound.Q
	                AND (#iqa_TrackingData[#si_PositionToUpdate] <> 0
	                AND #iqa_TrackingData[#si_PositionToUpdate] <> #si_LastUpdatedGIN)
	                AND NOT #sx_ParcelWaitEnable)
	            THEN
	                IF (#iqa_TrackingData[#si_PositionToUpdate] > 0)
	                THEN
	                    IF ("DB_GIN".GIN[#iqa_TrackingData[#si_PositionToUpdate]].General.Lost = FALSE)
	                    THEN
	                        "DB_GIN".GIN[#iqa_TrackingData[#si_PositionToUpdate]].General.Lost := TRUE;
	                        "FC_Fifo"(ic_Mode := 'W',
	                                  qUDT_Status => #sUDT_LostGINFIFOStatus,
	                                  qx_Error => #sx_LostGINFIFOError,
	                                  qx_Warning => #sx_LostGINFIFOWarning,
	                                  iqv_Data := #iqa_TrackingData[#si_PositionToUpdate],
	                                  iqUDT_FifoHeader := #iqUDT_FifoHeader,
	                                  iqv_DataBuffer := #iqa_FifoData);

	                        // Update statistics
	                        #ss_LostParcelsCounters.Total += 1;
	                        #ss_LostParcelsCounters.DoubleData += 1;

	                        ////////////////////

	                        IF #iqa_TrackingData[#si_PositionToUpdate] >= 1000 THEN
	                            #ss_LostValidParcelsCounters.Total += 1;
	                            #ss_LostValidParcelsCounters.DoubleData += 1;
	                        END_IF;

	                        ////////////////
	                        //
	                    END_IF;
	                END_IF;

	                // Generate GIN
	                #sx_GenerateGIN := TRUE;
	                #si_UnknownParcelsCounters.LostParcelFound += 1;

	                (*Second data has been found during data update. Situation can occur when search window is too short
	                  and the data is shifted. In that case found GIN will be marked as a lost one.*)
	            ELSIF (#sR_TRIG_PositiveDataFound.Q
	                AND #sx_ParcelDetected
	                AND #iqa_TrackingData[#si_PositionToUpdate] <> #si_GINToWrite)
	            THEN
	                // Mark GIN as a lost one
	                IF ("DB_GIN".GIN[#iqa_TrackingData[#si_PositionToUpdate]].General.Lost = FALSE)
	                THEN
	                    "DB_GIN".GIN[#iqa_TrackingData[#si_PositionToUpdate]].General.Lost := TRUE;
	                    "FC_Fifo"(ic_Mode := 'W',
	                              qUDT_Status => #sUDT_LostGINFIFOStatus,
	                              qx_Error => #sx_LostGINFIFOError,
	                              qx_Warning => #sx_LostGINFIFOWarning,
	                              iqv_Data := #iqa_TrackingData[#si_PositionToUpdate],
	                              iqUDT_FifoHeader := #iqUDT_FifoHeader,
	                              iqv_DataBuffer := #iqa_FifoData);

	                    // Update statistics
	                    #ss_LostParcelsCounters.Total += 1;
	                    #ss_LostParcelsCounters.DoubleData += 1;

	                    ////////////////////

	                    IF #iqa_TrackingData[#si_PositionToUpdate] >= 1000 THEN
	                        #ss_LostValidParcelsCounters.Total += 1;
	                        #ss_LostValidParcelsCounters.DoubleData += 1;
	                    END_IF;

	                    ////////////////
	                END_IF;
	            END_IF;

	        END_REGION

	        REGION 10.5 – GIN generator

	            (*Used to generate new GIN. If the PEC position is a generation point, the number is taken from an internal GIN range.
	              If it's not, then GIN is taken from a global unknown GIN range.*)

	            IF (#sx_GenerateGIN)
	            THEN
	                // Generation point.
	                IF (#iUDT_PECUpdateConfiguration.GenerationPoint)
	                THEN
	                    // Generate GIN from a valid GIN range.
	                    IF (#ss_ValidGINRange.GIN <= #ss_ValidGINRange.End)
	                    THEN
	                        #si_GINToWrite := #ss_ValidGINRange.GIN;
	                        #ss_ValidGINRange.GIN += 1;
	                    ELSE
	                        #si_GINToWrite := #ss_ValidGINRange.Start;
	                        #ss_ValidGINRange.GIN := #ss_ValidGINRange.Start + 1;
	                    END_IF;
	                    // Unknown GIN generator.
	                ELSE
	                    // Generate GIN from a unknown GIN range.
	                    IF (#iqUDT_UnknownGINRange.GIN <= #iqUDT_UnknownGINRange.End)
	                    THEN
	                        #si_GINToWrite := #iqUDT_UnknownGINRange.GIN;
	                        #iqUDT_UnknownGINRange.GIN += 1;
	                    ELSE
	                        #si_GINToWrite := #iqUDT_UnknownGINRange.Start;
	                        #iqUDT_UnknownGINRange.GIN := #iqUDT_UnknownGINRange.Start + 1;
	                    END_IF;

	                    // Unknwn parcels statistics.
	                    #si_UnknownParcelsCounters.Total += 1;
	                END_IF;

	                // Reset generte GIN command.
	                #sx_GenerateGIN := FALSE;

	                // GIN record is cleared with configured default GIN record while it's generated.
	                "DB_GIN".GIN[#si_GINToWrite] := "DB_GINDefault".GIN[#iUDT_PECUpdateConfiguration.DefaultGIN];
	            END_IF;

	            #qi_GINwrite := #si_GINToWrite;

	        END_REGION


	        REGION 10.6 – PEC position data update

	            (*While parcel is detected, calculated GIN is written into the PEC position record.
	              If not, then the record is cleared with 0. Negative GIN is ignored or deleted, depending on configuration.*)

	            IF (#sx_ParcelDetected)
	            THEN

	                "FC_WriteGIN"(ii_GIN := #si_GINToWrite,
	                              ii_PositionToWrite := #si_PositionToUpdate,
	                              ii_NumberOfPositions := 1,
	                              ix_Direction := TRUE,
	                              iqa_TrackingData := #iqa_TrackingData);

	            ELSE
	                IF (#iqa_TrackingData[#si_PositionToUpdate] > 0
	                    OR #iUDT_PECUpdateConfiguration.NegativeGINDelete)
	                THEN

	                    "FC_WriteGIN"(ii_GIN := #ci_ZeroGIN,
	                                  ii_PositionToWrite := #si_PositionToUpdate,
	                                  ii_NumberOfPositions := 1,
	                                  ix_Direction := TRUE,
	                                  iqa_TrackingData := #iqa_TrackingData);

	                END_IF;
	            END_IF;

	        END_REGION

	        REGION 10.7 – Parcel waiting logic

	            (*Parcel waiting logic is used to wait for the photoeye signal for a search window distance.*)
	            IF (#sx_ParcelWaitEnable)
	            THEN
	                // Counting parcel wait distance depending on conveyor running direction if not detected.
	                IF (NOT #sx_ParcelDetected)
	                THEN
	                    IF (#si_Direction = 1)
	                    THEN
	                        #si_ParcelWaitDistance += 1;
	                    ELSE
	                        #si_ParcelWaitDistance -= 1;
	                    END_IF;

	                    // Parcel detected - stop waiting, use found GIN to update.
	                ELSE
	                    // PEC/Data deviation acquisition
	                    #ss_PECDataDeviation.Last := #si_ParcelWaitDistance;
	                    #ss_PECDataDeviation.GIN := #si_GINToWrite;
	                    #ss_PECDataDeviation.Sum += ABS(#ss_PECDataDeviation.Last);
	                    #ss_PECDataDeviation.Nr += 1;


	                    // Parcel aligned statistics
	                    IF (#ss_PECDataDeviation.Last > ABS(#si_Displacement - 1))
	                    THEN
	                        #ss_AlignedParcelsCounters.Total += 1;
	                        #ss_AlignedParcelsCounters.DataNoPEC += 1;
	                    END_IF;

	                    // Parcel waiting logic reset.
	                    #sx_ParcelWaitEnable := FALSE;
	                    #si_ParcelWaitDistance := 0;
	                END_IF;
	            END_IF;

	            // Parcel not found in a search window - stop waiting, mark found GIN as a lost one.
	            IF (ABS(#si_ParcelWaitDistance) = #si_SearchWindow)
	                AND (#si_GINToWrite > 0)
	            THEN
	                // Parcel lost
	                IF "DB_GIN".GIN[#si_GINToWrite].General.Lost = FALSE THEN
	                    "DB_GIN".GIN[#si_GINToWrite].General.Lost := TRUE;
	                    "FC_Fifo"(ic_Mode := 'W',
	                              qUDT_Status => #sUDT_LostGINFIFOStatus,
	                              qx_Error => #sx_LostGINFIFOError,
	                              qx_Warning => #sx_LostGINFIFOWarning,
	                              iqv_Data := #si_GINToWrite,
	                              iqUDT_FifoHeader := #iqUDT_FifoHeader,
	                              iqv_DataBuffer := #iqa_FifoData);

	                    // Parcel waiting logic reset.
	                    #si_ParcelWaitDistance := 0;
	                    #sx_ParcelWaitEnable := FALSE;

	                    // Lost parcels ina  row counter.
	                    #si_LostParcelsInARow += 1;

	                    // Update statistics.
	                    #ss_LostParcelsCounters.Total += 1;
	                    #ss_LostParcelsCounters.ParcelNotFound += 1;

	                    ////////////////////

	                    IF #si_GINToWrite >= 1000 THEN
	                        #ss_LostValidParcelsCounters.Total += 1;
	                        #ss_LostValidParcelsCounters.ParcelNotFound += 1;
	                    END_IF;

	                    ////////////////
	                    //
	                END_IF;

	            END_IF;

	            // Reset monitoring in case of going backwards.
	            IF (#si_ParcelWaitDistance = 0
	                AND NOT #sx_ParcelDetected
	                AND #sx_InvalidDirection)
	            THEN
	                #sx_ParcelWaitEnable := FALSE;
	            END_IF;

	            #sx_InvalidDirection := ((#si_Direction = 1
	            AND #si_ParcelWaitDistance < 0)
	            OR (#si_Direction = -1
	            AND #si_ParcelWaitDistance > 0));

	        END_REGION

	        REGION 10.8 – Last updated GIN

	            (*Last updated GIN to avoid processing the same data.*)
	            IF (#sR_TRIG_DataFound.Q)
	            THEN
	                #si_LastUpdatedGIN := #iqa_TrackingData[#si_PositionToUpdate];
	            END_IF;

	        END_REGION

	        REGION 10.8 – Update displacement

	            #si_Displacement := #si_Displacement - #si_Direction;

	        END_REGION

	    END_WHILE;

	END_REGION

	REGION 11 – Length measurement



	    (*Length and gap measurements can be enabled via PEC update configuration*)
	    #sFB_LengthMeasurement(ii_PECPosition := #si_PECPosition,
	                           ii_Displacement := #iqUDT_ConveyorInterface.Displacement,
	                           ix_LengthMeasurementEnable := #iUDT_PECUpdateConfiguration.ParcelLengthMeasurement OR #sx_LengthMeasurementEnable,
	                           ix_GapMeasurementEnable := #iUDT_PECUpdateConfiguration.GapLengthMeasurement,
	                           iqa_TrackingData := #iqa_TrackingData);

	    IF #iqa_TrackingData[#si_PECPosition] > 0
	        AND #iqa_TrackingData[#si_PECPosition] >= #iqUDT_UnknownGINRange.Start
	        AND #iqa_TrackingData[#si_PECPosition] <= #iqUDT_UnknownGINRange.End
	    THEN

	        #sx_LengthMeasurementEnable := "DB_GIN".GIN[#iqa_TrackingData[#si_PECPosition]].General.Length = 0;
	    ELSE

	        #sx_LengthMeasurementEnable := FALSE;

	    END_IF;

	END_REGION

	REGION 12 – Teaching done

	    // Average slip calculation
	    #si_AverageSlip := #ss_PECDataDeviation.Sum / #ss_PECDataDeviation.Nr;
	    #si_CalculatedLengthCorrection := DINT_TO_INT(#iUDT_ConveyorCommonConfiguration.LengthCorrection) + #si_AverageSlip * 10;
	    IF (#sx_TeachingMode                                                                                                            // Teaching mode enabled
	        AND #si_NumberOfTeachedParcels = #iUDT_PECUpdateConfiguration.NrOfTeachParcels)                                                 // Number of teaching parcels equal to the preset one                                                                                                                                                              // Teaching mode enabled ("sx_TeachMode")
	    THEN

	        #si_CalculatedLengthCorrection := DINT_TO_INT(#iUDT_ConveyorCommonConfiguration.LengthCorrection) + #si_AverageSlip * 10;
	        #sx_TeachingMode := FALSE;
	        #si_NumberOfTeachedParcels := 0;

	    END_IF;

	END_REGION

	REGION 13 – Performance

	    (*Performnce is a percentage ratio between number of lost parcels and total number of data, used to monitor data update efficiency.*)

	    IF (#sdi_TotalNumberOfData >= #ss_LostParcelsCounters.Total
	        AND #sdi_TotalNumberOfData > 0)
	    THEN
	        #slr_Performance := 100.0 - INT_TO_LREAL(#ss_LostParcelsCounters.Total) / #sdi_TotalNumberOfData * 100.0;
	    END_IF;

	    // Warning is generated if performance drops below 80%.
	    #qUDT_Status.LowPerformance := #slr_Performance < 80;

	END_REGION

	REGION 14 – Reset statistics

	    // Statistics are reset if reset signal is given.
	    IF #iqUDT_ConveyorInterface.ResetStatistics
	    THEN
	        #sdi_TotalNumberOfParcels := 0;
	        #ss_AlignedParcelsCounters.Total := 0;
	        #ss_AlignedParcelsCounters.PECNoData := 0;
	        #ss_AlignedParcelsCounters.DataNoPEC := 0;
	        #ss_LostParcelsCounters.Total := 0;
	        #ss_LostParcelsCounters.DoubleData := 0;
	        #ss_LostParcelsCounters.ParcelNotFound := 0;
	        #ss_LostValidParcelsCounters.Total := 0;
	        #ss_LostValidParcelsCounters.DoubleData := 0;
	        #ss_LostValidParcelsCounters.ParcelNotFound := 0;
	        #sdi_TotalNumberOfData := 0;
	        #si_UnknownParcelsCounters.Total := 0;
	        #si_UnknownParcelsCounters.LostParcelFound := 0;
	        #si_UnknownParcelsCounters.DataNotFound := 0;
	        #ss_PECDataDeviation.Sum := 0;
	        #ss_PECDataDeviation.Nr := 0;
	        #slr_Performance := 100;

	    END_IF;

	END_REGION

	REGION 15 – Too many lost parcels error

	    (*Error is generated if too many parcels will is marked as a lost one in a row*)
	    IF (#si_LostParcelsInARow >= #iUDT_PECUpdateConfiguration.MaxLost)
	    THEN
	        #qUDT_Status.TooManyLost := TRUE;
	    END_IF;

	END_REGION

	REGION 16 – Statistics

	    // Too many lost
	    #sR_TRIG_TooManyLost(CLK := #qUDT_Status.TooManyLost);
	    IF #qUDT_Status.TooManyLost
	        OR #iqUDT_ConveyorInterface.ResetStatistics
	    THEN
	        "FC_Statistics"(ix_Reset := #iqUDT_ConveyorInterface.ResetStatistics,
	                        ix_Activate := #qUDT_Status.TooManyLost,
	                        ix_RTrigActivate := #sR_TRIG_TooManyLost.Q,
	                        iqUDT_Statistics := #iqUDT_Statistics.TooManyLost);
	    END_IF;

	    // Total number of parcels
	    #iqUDT_Statistics.TotalNrOfParcels := #sdi_TotalNumberOfParcels;

	END_REGION

	REGION 17 – Internal tracking warning and error

	    // Internal tracking warning
	    IF (#qUDT_Status.LowPerformance
	        OR #sx_LostGINFIFOWarning)
	    THEN
	        #iqUDT_ConveyorInterface.InternalWarningTracking := TRUE;
	    END_IF;

	    // Internal tracking error
	    IF #qUDT_Status.TooManyLost
	    THEN
	        #iqUDT_ConveyorInterface.InternalErrorTracking := TRUE;
	    END_IF;

	    // Configuration error
	    IF (#sx_InvalidDisplacement
	        OR #sx_InvalidGINRange
	        OR #sx_InvalidSearchWindow)
	    THEN
	        #iqUDT_ConveyorInterface.ConfigurationError := TRUE;
	    END_IF;

	END_REGION
END_FUNCTION_BLOCK

FUNCTION_BLOCK "FB_VSULift"
TITLE = FB_VerticalSwitch
{ S7_Optimized_Access := 'TRUE' }
AUTHOR : MHSE
FAMILY : Equipment
VERSION : 3.0
// ATTRIBUTES
// AUTO_NUMBER = True
// BLOCK_NUMBER = 258
// END_ATTRIBUTES
//Function block to control vertical switch unit.
   VAR_INPUT
      iUDT_VSUConfig { ExternalAccessible := 'False'; ExternalVisible := 'False'; ExternalWritable := 'False'} : "UDT_VSULiftConfiguration";   // VSU Configuration structure
      ix_SafetyOk { ExternalAccessible := 'False'; ExternalVisible := 'False'; ExternalWritable := 'False'} : Bool;   // TRUE when Safety Circuit of the Conveyor is healthy
      ix_BeltTear1 { ExternalAccessible := 'False'; ExternalVisible := 'False'; ExternalWritable := 'False'} : Bool;   // TRUE when Belt tear switch 1 is ok
      ix_BeltTear2 { ExternalAccessible := 'False'; ExternalVisible := 'False'; ExternalWritable := 'False'} : Bool;   // TRUE when Belt tear switch 2 is ok
      ix_MaintSupport1 { ExternalAccessible := 'False'; ExternalVisible := 'False'; ExternalWritable := 'False'} : Bool;   // TRUE when lift maintenance support 1 is retracted
      ix_MaintSupport2 { ExternalAccessible := 'False'; ExternalVisible := 'False'; ExternalWritable := 'False'} : Bool;   // TRUE when lift maintenance support 2 is retracted
      ix_PosUp { ExternalAccessible := 'False'; ExternalVisible := 'False'; ExternalWritable := 'False'} : Bool;   // TRUE when position sensor is covered
      ix_PosDown { ExternalAccessible := 'False'; ExternalVisible := 'False'; ExternalWritable := 'False'} : Bool;   // TRUE when position sensor is covered
      ix_PECGapEnd { ExternalAccessible := 'False'; ExternalVisible := 'False'; ExternalWritable := 'False'} : Bool;   // TRUE when PEC Jamdetection going up is not blocked
      ix_PECGapBegin { ExternalAccessible := 'False'; ExternalVisible := 'False'; ExternalWritable := 'False'} : Bool;   // TRUE when PEC Jamdetection going down is not blocked
      ix_LimitSwitchUp { ExternalAccessible := 'False'; ExternalVisible := 'False'; ExternalWritable := 'False'} : Bool;   // TRUE when limit position is overrun
      ix_LimitSwitchDown { ExternalAccessible := 'False'; ExternalVisible := 'False'; ExternalWritable := 'False'} : Bool;   // TRUE when limit position is overrun
      ix_SafetyDoorDiagDown { ExternalAccessible := 'False'; ExternalVisible := 'False'; ExternalWritable := 'False'} : Bool;   // TRUE safety door diagnosis ok (Down)
      ix_SafetyDoorDiagUp { ExternalAccessible := 'False'; ExternalVisible := 'False'; ExternalWritable := 'False'} : Bool;   // TRUE safety door diagnosis ok (Up)
      ix_LCPAutoMode { ExternalAccessible := 'False'; ExternalVisible := 'False'; ExternalWritable := 'False'} : Bool;   // TRUE when LocalControlPanel switch Automatic is on
      ix_LCPManualMode { ExternalAccessible := 'False'; ExternalVisible := 'False'; ExternalWritable := 'False'} : Bool;   // TRUE when LocalControlPanel switch Manual is on
      ix_LCPStop { ExternalAccessible := 'False'; ExternalVisible := 'False'; ExternalWritable := 'False'} : Bool;   // TRUE when LocalControlPanel switch Stop is on
      ix_LCPDown { ExternalAccessible := 'False'; ExternalVisible := 'False'; ExternalWritable := 'False'} : Bool;   // TRUE when LocalControlPanel switch Down is on
      ix_LCPUp { ExternalAccessible := 'False'; ExternalVisible := 'False'; ExternalWritable := 'False'} : Bool;   // TRUE when LocalControlPanel switch Up is on
      ix_LCPRef { ExternalAccessible := 'False'; ExternalVisible := 'False'; ExternalWritable := 'False'} : Bool;   // TRUE when LocalControlPanel switch Refference is on
      ix_TransportIdle { ExternalAccessible := 'False'; ExternalVisible := 'False'; ExternalWritable := 'False'} : Bool;   // TRUE when lift block signals transport is idle
      ix_HardwareOk { ExternalAccessible := 'False'; ExternalVisible := 'False'; ExternalWritable := 'False'} : Bool;   // TRUE when  hardware is Ok
      ix_MaintenanceSwitchUp { ExternalAccessible := 'False'; ExternalVisible := 'False'; ExternalWritable := 'False'} : Bool;   // TRUE when Maintenance Switch is turned  on
      ix_MainContactorFeedback { ExternalAccessible := 'False'; ExternalVisible := 'False'; ExternalWritable := 'False'} : Bool;   // TRUE when Main Contactor is OK
      ix_OverTempBrakingResistor { ExternalAccessible := 'False'; ExternalVisible := 'False'; ExternalWritable := 'False'} : Bool;   // TRUE when Over Temperature Braking Resisitor is OK
   END_VAR

   VAR_OUTPUT
      qUDT_HMIStatus { ExternalAccessible := 'False'; ExternalVisible := 'False'; ExternalWritable := 'False'} : "UDT_VSULiftStatus";   // HMI status structure
      qUDT_Status { ExternalAccessible := 'False'; ExternalVisible := 'False'; ExternalWritable := 'False'} : "UDT_CommonStatus";   // Common status structure
      qx_MainContactorOn { ExternalAccessible := 'False'; ExternalVisible := 'False'; ExternalWritable := 'False'} : Bool;   // Main Contactor On
   END_VAR

   VAR_IN_OUT
      iqUDT_EquipmentControl : "UDT_EquipmentControl";   // Equipment control structure
      iqUDT_VSUCommand : "UDT_VSUCommand";   // VSU HMI Command structure
      iqUDT_VSUInterface : "UDT_VSUInterface";   // Interface between VSU and VFD
      iqUDT_Statistics : "UDT_VSULiftStatistics";   // Statistics structure
   END_VAR

   VAR
      sUDT_HMIStatus { ExternalAccessible := 'False'; ExternalVisible := 'False'; ExternalWritable := 'False'; S7_SetPoint := 'False'} : "UDT_VSULiftStatus";   // HMI status structure
      sUDT_StatusOld { ExternalAccessible := 'False'; ExternalVisible := 'False'; ExternalWritable := 'False'; S7_SetPoint := 'False'} : "UDT_CommonStatus";   // Common status structure
      sUDT_Status { ExternalAccessible := 'False'; ExternalVisible := 'False'; ExternalWritable := 'False'; S7_SetPoint := 'False'} : "UDT_CommonStatus";   // Common status structure
      sFB_PECEoSFiltered { ExternalAccessible := 'False'; ExternalVisible := 'False'; ExternalWritable := 'False'; S7_SetPoint := 'False'} : "FB_TimerOnOffDelay";   // Filtering end of section photo eye signal
      sFB_PEC_GapEndFiltered { ExternalAccessible := 'False'; ExternalVisible := 'False'; ExternalWritable := 'False'; S7_SetPoint := 'False'} : "FB_TimerOnOffDelay";   // Filtering upper jam photo eye signal
      sFB_PEC_GapBeginFiltered { ExternalAccessible := 'False'; ExternalVisible := 'False'; ExternalWritable := 'False'; S7_SetPoint := 'False'} : "FB_TimerOnOffDelay";   // Filtering lower jam photo eye signal
      sFB_JogEnable { ExternalAccessible := 'False'; ExternalVisible := 'False'; ExternalWritable := 'False'; S7_SetPoint := 'False'} : "FB_TimerOnOffDelay";   // Filtering lower jam photo eye signal
      sFB_MaxStopTime { ExternalAccessible := 'False'; ExternalVisible := 'False'; ExternalWritable := 'False'; S7_SetPoint := 'False'} : "FB_TimerOnOffDelay";   // Timer for maximum stopping time
      sR_TRIG_ManualMode {InstructionName := 'R_TRIG'; LibVersion := '1.0'; ExternalAccessible := 'False'; ExternalVisible := 'False'; ExternalWritable := 'False'; S7_SetPoint := 'False'} : R_TRIG;   // Rising edge trigger manual mode
      sR_TRIG_ManualJogUp {InstructionName := 'R_TRIG'; LibVersion := '1.0'; ExternalAccessible := 'False'; ExternalVisible := 'False'; ExternalWritable := 'False'; S7_SetPoint := 'False'} : R_TRIG;   // Rising edge trigger manual jog mode command
      sR_TRIG_ManualJogDown {InstructionName := 'R_TRIG'; LibVersion := '1.0'; ExternalAccessible := 'False'; ExternalVisible := 'False'; ExternalWritable := 'False'; S7_SetPoint := 'False'} : R_TRIG;   // Rising edge trigger manual jog mode command
      sR_TRIG_DownTime {InstructionName := 'R_TRIG'; LibVersion := '1.0'; ExternalAccessible := 'False'; ExternalVisible := 'False'; ExternalWritable := 'False'; S7_SetPoint := 'False'} : R_TRIG;   // Rising edge trigger VSU is stopped
      sR_TRIG_Error {InstructionName := 'R_TRIG'; LibVersion := '1.0'; ExternalAccessible := 'False'; ExternalVisible := 'False'; ExternalWritable := 'False'; S7_SetPoint := 'False'} : R_TRIG;   // Rising edge trigger for Error
      sR_TRIG_GapExit_Error {InstructionName := 'R_TRIG'; LibVersion := '1.0'; ExternalAccessible := 'False'; ExternalVisible := 'False'; ExternalWritable := 'False'; S7_SetPoint := 'False'} : R_TRIG;   // Rising edge trigger for Exit gap check error
      sR_TRIG_GapEntry_Error {InstructionName := 'R_TRIG'; LibVersion := '1.0'; ExternalAccessible := 'False'; ExternalVisible := 'False'; ExternalWritable := 'False'; S7_SetPoint := 'False'} : R_TRIG;   // Rising edge trigger for Entry gap check error
      sR_TRIG_BeltTear1 {InstructionName := 'R_TRIG'; LibVersion := '1.0'; ExternalAccessible := 'False'; ExternalVisible := 'False'; ExternalWritable := 'False'; S7_SetPoint := 'False'} : R_TRIG;   // Rising edge trigger for Belt tear 1 detected
      sR_TRIG_BeltTear2 {InstructionName := 'R_TRIG'; LibVersion := '1.0'; ExternalAccessible := 'False'; ExternalVisible := 'False'; ExternalWritable := 'False'; S7_SetPoint := 'False'} : R_TRIG;   // Rising edge trigger for Belt tear 2 detected
      sR_TRIG_MaintSupport1Err {InstructionName := 'R_TRIG'; LibVersion := '1.0'; ExternalAccessible := 'False'; ExternalVisible := 'False'; ExternalWritable := 'False'; S7_SetPoint := 'False'} : R_TRIG;   // Rising edge trigger for Maintenace support 1 extracted
      sR_TRIG_MaintSupport2Err {InstructionName := 'R_TRIG'; LibVersion := '1.0'; ExternalAccessible := 'False'; ExternalVisible := 'False'; ExternalWritable := 'False'; S7_SetPoint := 'False'} : R_TRIG;   // Rising edge trigger for Maintenace support 2 extracted
      sR_TRIG_UpperPositionErr {InstructionName := 'R_TRIG'; LibVersion := '1.0'; ExternalAccessible := 'False'; ExternalVisible := 'False'; ExternalWritable := 'False'; S7_SetPoint := 'False'} : R_TRIG;   // Rising edge trigger for Upper position overrun
      sR_TRIG_LowerPositionErr {InstructionName := 'R_TRIG'; LibVersion := '1.0'; ExternalAccessible := 'False'; ExternalVisible := 'False'; ExternalWritable := 'False'; S7_SetPoint := 'False'} : R_TRIG;   // Rising edge trigger for Lower position overrun
      sR_TRIG_SafetyDoorErr {InstructionName := 'R_TRIG'; LibVersion := '1.0'; ExternalAccessible := 'False'; ExternalVisible := 'False'; ExternalWritable := 'False'; S7_SetPoint := 'False'} : R_TRIG;   // Rising edge trigger for Safety door diagnostic fault
      sR_TRIG_Direction_Error {InstructionName := 'R_TRIG'; LibVersion := '1.0'; ExternalAccessible := 'False'; ExternalVisible := 'False'; ExternalWritable := 'False'; S7_SetPoint := 'False'} : R_TRIG;   // Rising edge trigger for Direction error
      sR_TRIG_UpTime {InstructionName := 'R_TRIG'; LibVersion := '1.0'; ExternalAccessible := 'False'; ExternalVisible := 'False'; ExternalWritable := 'False'; S7_SetPoint := 'False'} : R_TRIG;   // Rising edge trigger VSU is running automatic
      sR_TRIG_GOReference {InstructionName := 'R_TRIG'; LibVersion := '1.0'; ExternalAccessible := 'False'; ExternalVisible := 'False'; ExternalWritable := 'False'; S7_SetPoint := 'False'} : R_TRIG;   // Rising edge trigger for VFD to do reference run
      sR_TRIG_Referenced {InstructionName := 'R_TRIG'; LibVersion := '1.0'; ExternalAccessible := 'False'; ExternalVisible := 'False'; ExternalWritable := 'False'; S7_SetPoint := 'False'} : R_TRIG;   // Rising edge trigger VFD refferenced
      sR_TRIG_TIPLeavingVSU {InstructionName := 'R_TRIG'; LibVersion := '1.0'; ExternalAccessible := 'False'; ExternalVisible := 'False'; ExternalWritable := 'False'; S7_SetPoint := 'False'} : R_TRIG;   // Rising edge trigger TIP VSU Conveyor
      sF_TRIG_TIPLeavingVSU {InstructionName := 'F_TRIG'; LibVersion := '1.0'; ExternalAccessible := 'False'; ExternalVisible := 'False'; ExternalWritable := 'False'; S7_SetPoint := 'False'} : F_TRIG;   // Falling edge trigger TIP VSU Conveyor
      sR_TRIG_RestartFromError {InstructionName := 'R_TRIG'; LibVersion := '1.0'; ExternalAccessible := 'False'; ExternalVisible := 'False'; ExternalWritable := 'False'; S7_SetPoint := 'False'} : R_TRIG;   // Rising edge trigger Restart from error
   END_VAR
   VAR RETAIN
      sdi_RunEmpty { ExternalAccessible := 'False'; ExternalVisible := 'False'; ExternalWritable := 'False'} : DInt;   // Calculation run empty distance
   END_VAR
   VAR
      si_Position { ExternalAccessible := 'False'; ExternalVisible := 'False'; ExternalWritable := 'False'} : Int;   // Position from Decisionpoint
      si_RequiredGap { ExternalAccessible := 'False'; ExternalVisible := 'False'; ExternalWritable := 'False'} : Int;   // Required gap in front of VSU
   END_VAR
   VAR RETAIN
      si_UpperHeadToHead { ExternalAccessible := 'False'; ExternalVisible := 'False'; ExternalWritable := 'False'} : Int;   // Gap calculation Head To Head upper conveyor
      si_UpperGap { ExternalAccessible := 'False'; ExternalVisible := 'False'; ExternalWritable := 'False'} : Int;   // Gap calculation upper outfeed conveyor
      si_LowerHeadToHead { ExternalAccessible := 'False'; ExternalVisible := 'False'; ExternalWritable := 'False'} : Int;   // Gap calculation Head To Head lower conveyor
      si_LowerGap { ExternalAccessible := 'False'; ExternalVisible := 'False'; ExternalWritable := 'False'} : Int;   // Gap calculation lower outfeed conveyor
      si_UpJamDisplacement { ExternalAccessible := 'False'; ExternalVisible := 'False'; ExternalWritable := 'False'} : Int;   // Auxiliary variable to calculate displacement when PEC is blocked
      si_LowJamDisplacement { ExternalAccessible := 'False'; ExternalVisible := 'False'; ExternalWritable := 'False'} : Int;   // Auxiliary variable to calculate displacement when PEC is blocked
   END_VAR
   VAR
      si_DefaultPosition { ExternalAccessible := 'False'; ExternalVisible := 'False'; ExternalWritable := 'False'} : Int;   // Auxiliary variable to set default position
      sx_StartReceived { ExternalAccessible := 'False'; ExternalVisible := 'False'; ExternalWritable := 'False'} : Bool;   // Start command received from system
      sx_PEC_EoSFiltered { ExternalAccessible := 'False'; ExternalVisible := 'False'; ExternalWritable := 'False'} : Bool;   // End of section photo eye filtered
      sx_PEC_UpOutFiltered { ExternalAccessible := 'False'; ExternalVisible := 'False'; ExternalWritable := 'False'} : Bool;   // Upper outfeed photo eye filtered
      sx_PEC_LowOutFiltered { ExternalAccessible := 'False'; ExternalVisible := 'False'; ExternalWritable := 'False'} : Bool;   // Lower outfeed photo eye filtered
      sx_PEC_GapEnd { ExternalAccessible := 'False'; ExternalVisible := 'False'; ExternalWritable := 'False'} : Bool;   // Upper jam photo eye filtered
      sx_PEC_GapBegin { ExternalAccessible := 'False'; ExternalVisible := 'False'; ExternalWritable := 'False'} : Bool;   // Lower jam photo eye filtered
      sx_Ready { ExternalAccessible := 'False'; ExternalVisible := 'False'; ExternalWritable := 'False'} : Bool;   // Conveyor Ready to operate in Automatic mode
      sx_AutomaticActive { ExternalAccessible := 'False'; ExternalVisible := 'False'; ExternalWritable := 'False'} : Bool;   // Running in automatic
      sx_SemiAutomatic { ExternalAccessible := 'False'; ExternalVisible := 'False'; ExternalWritable := 'False'} : Bool;   // Running in semi automatic
      sx_PositionAfterRef { ExternalAccessible := 'False'; ExternalVisible := 'False'; ExternalWritable := 'False'} : Bool;   // After reffer
      sx_PreStartManual { ExternalAccessible := 'False'; ExternalVisible := 'False'; ExternalWritable := 'False'} : Bool;   // Pre conditions to run conveyor in manual mode
      sx_ManualModeActive { ExternalAccessible := 'False'; ExternalVisible := 'False'; ExternalWritable := 'False'} : Bool;   // Manual mode active
      sx_Stopping { ExternalAccessible := 'False'; ExternalVisible := 'False'; ExternalWritable := 'False'} : Bool;   // Stopping is active, first reach position
      sx_SwitchEnable { ExternalAccessible := 'False'; ExternalVisible := 'False'; ExternalWritable := 'False'} : Bool;   // Switching conditions
      sx_UpRequest { ExternalAccessible := 'False'; ExternalVisible := 'False'; ExternalWritable := 'False'} : Bool;   // Request upper outfeed position for actual parcel
      sx_DownRequest { ExternalAccessible := 'False'; ExternalVisible := 'False'; ExternalWritable := 'False'} : Bool;   // Request lower outfeed position for actual parcel
      sx_ActualPositionUP { ExternalAccessible := 'False'; ExternalVisible := 'False'; ExternalWritable := 'False'} : Bool;   // Actual position is up
      sx_ActualPositionDown { ExternalAccessible := 'False'; ExternalVisible := 'False'; ExternalWritable := 'False'} : Bool;   //   Actual position is down
      sx_GappingUpper { ExternalAccessible := 'False'; ExternalVisible := 'False'; ExternalWritable := 'False'} : Bool;   //   Gapping upper outfeed is active
      sx_GappingLower { ExternalAccessible := 'False'; ExternalVisible := 'False'; ExternalWritable := 'False'} : Bool;   //   Gapping lower outfeed is active
      sx_CombinedJogUp { ExternalAccessible := 'False'; ExternalVisible := 'False'; ExternalWritable := 'False'} : Bool;   //   Combined signal of jogging buttons
      sx_CombinedJogDown { ExternalAccessible := 'False'; ExternalVisible := 'False'; ExternalWritable := 'False'} : Bool;   //   Combined signal of jogging buttons
      sx_RestartFromError { ExternalAccessible := 'False'; ExternalVisible := 'False'; ExternalWritable := 'False'} : Bool;   //   After an error has occurred the action to be done before resuming normal operation
      sx_StopInfeed { ExternalAccessible := 'False'; ExternalVisible := 'False'; ExternalWritable := 'False'} : Bool;   //   Stop infeed conveyor
      sx_Jog { ExternalAccessible := 'False'; ExternalVisible := 'False'; ExternalWritable := 'False'} : Bool;   //   Off delayed signal Jogging was activated
      sx_ConfigurationError { ExternalAccessible := 'False'; ExternalVisible := 'False'; ExternalWritable := 'False'} : Bool;   //   Commissioning: configuration of parameters is wrong
   END_VAR

   VAR_TEMP
      tr_req : Real;
   END_VAR

   VAR CONSTANT
      ci_PositionUp : Int := 2;   //   Value for UP Position
      ci_PositionDown : Int := 1;   //   Value for DOWN Position
      ci_PositionDefault : Int := 99;   //   Value for DEFAULT Position
   END_VAR


BEGIN
	(*

	----------------------------------------------------------------------------------------

	Version history:
	Date        | Version   | Author        | Remark
	----------------------------------------------------------------------------------------
	19/10/2023  | 1.0       | F.Baten       | FB_VSULift: Branched version of FB_VSU for Lift application without gapping and tracking
	19/10/2023  | 1.1       | J.Majer       | Clear unused functions and adding belt tear, gap check, up&down limit switch, lifting carriage supports inputs with statistics and status
	14/06/2024  | 1.2       | R. Pieczonka  | Added new errors
	*)

	REGION 1 - Initial

	    REGION 1.1 - First PLC cycle

	        IF "DB_Memory".FirstScan
	        THEN
	            #sx_AutomaticActive := FALSE;                                               // switch of automatic active
	        END_IF;

	    END_REGION

	    REGION 1.2 - Triggers

	        // Detecting rising edge on manual mode Or from Equipment Control
	        #sR_TRIG_ManualMode(CLK := #sUDT_Status.Manual);

	        // Rising edge trigger running
	        #sR_TRIG_UpTime(CLK := #sx_AutomaticActive AND #sx_Ready);

	        // Detecting rising edge VSU stopped
	        #sR_TRIG_DownTime(CLK := #sx_AutomaticActive AND NOT #sx_Ready);

	        // Detecting rising edge on VSU error
	        #sR_TRIG_Error(CLK := #sUDT_Status.Error);

	        // Detecting rising edge on start of the restart from error sequence
	        #sR_TRIG_RestartFromError(CLK := #sx_RestartFromError);

	    END_REGION

	    REGION 1.3 - Filters

	        //Gap check end detection photo eye signal filtering
	        #sFB_PEC_GapEndFiltered(iudi_OnDelayTime := #iUDT_VSUConfig.PEC_GapEndOnDelay,
	                                iudi_OffDelayTime := #iUDT_VSUConfig.PEC_GapEndOffDelay,
	                                ix_SignalToDelay := #ix_PECGapEnd,
	                                ix_Enable := TRUE,
	                                qx_DelayedSignal => #sx_PEC_GapEnd);

	        //Gap check begin detection photo eye signal filtering
	        #sFB_PEC_GapBeginFiltered(iudi_OnDelayTime := #iUDT_VSUConfig.PEC_GapBeginOnDelay,
	                                  iudi_OffDelayTime := #iUDT_VSUConfig.PEC_GapBeginOffDelay,
	                                  ix_SignalToDelay := #ix_PECGapBegin,
	                                  ix_Enable := TRUE,
	                                  qx_DelayedSignal => #sx_PEC_GapBegin);

	        // Time to start without start warning while jogging
	        #sFB_JogEnable(iudi_OffDelayTime := #iUDT_VSUConfig.JogNoHornTime,
	                       ix_SignalToDelay := #sx_Jog);

	        // Maximum stopping time
	        #sFB_MaxStopTime(iudi_OnDelayTime := (#iUDT_VSUConfig.SwitchingTime + #iUDT_VSUConfig.SwitchingTime),
	                         ix_SignalToDelay := #sx_Stopping);
	    END_REGION

	    REGION 1.4 - Switching conditions

	        #sx_SwitchEnable :=                                                       // Enabling of direction switching
	        #ix_TransportIdle                                                         // No transfer in progress
	        AND #sx_PEC_GapBegin                                                      // entry gap sensor free
	        AND #sx_PEC_GapEnd                                                        // exit gap sensor free
	        AND #ix_BeltTear1                                                         // belt tear sensor 1 ok
	        AND #ix_BeltTear2                                                         // belt tear sensor 2 ok
	        AND #ix_MaintSupport1                                                     // Lift support extracted in automatic mode
	        AND #ix_MaintSupport1                                                     // Lift support extracted in automatic mode
	        AND NOT #ix_LimitSwitchUp                                                 // upper limit switch not overrun
	        AND NOT #ix_LimitSwitchDown                                               // lower limit switch not overrun
	        ;

	    END_REGION

	    REGION 1.5 - Position

	        #sx_ActualPositionUP :=                                                         // Set status bit lift in upper position
	        (#iqUDT_VSUInterface.PositionActual = #ci_PositionUp)                           // If actual position is equal to up
	        AND NOT #iqUDT_VSUInterface.Positioning                                         // And the positioning is not active
	        AND #ix_PosUp;                                                                  // And the position sensor signals

	        #sx_ActualPositionDown :=                                                       // Set bit lift in lower position
	        (#iqUDT_VSUInterface.PositionActual = #ci_PositionDown)                         // If actual position is equal to down
	        AND NOT #iqUDT_VSUInterface.Positioning                                         // And the positioning is not active
	        AND #ix_PosDown;                                                                // And the position sensor signals
	    END_REGION

	    REGION 1.6 - Check configuration
	        #si_DefaultPosition := #iUDT_VSUConfig.DefaultPosition;

	        IF #si_DefaultPosition <= 0
	        THEN
	            #si_DefaultPosition := #ci_PositionDown;

	        END_IF;
	    END_REGION
	END_REGION

	REGION 2 - Errors

	    REGION 2.1 - Reset errors

	        IF #iqUDT_EquipmentControl.Command.Reset                                       // Reset
	        THEN
	            // Gap check
	            IF #sUDT_HMIStatus.Specific.ExitGapErr                            // Exit gap check is active
	                AND (#sx_PEC_GapEnd OR #iqUDT_VSUInterface.PositionActual = #iqUDT_VSUInterface.PositionSetpoint)                                                      // Upper jam sensor is free
	            THEN
	                #sUDT_HMIStatus.Specific.ExitGapErr := FALSE;                 // reset error

	            END_IF;

	            IF #sUDT_HMIStatus.Specific.EntryGapErr                            // Entry gap check is active
	                AND (#sx_PEC_GapBegin OR #iqUDT_VSUInterface.PositionActual = #iqUDT_VSUInterface.PositionSetpoint)                                                   // Lower jam sensor is free
	            THEN
	                #sUDT_HMIStatus.Specific.EntryGapErr := FALSE;             // reset error

	            END_IF;

	            // Belt tear switch 1
	            IF #ix_BeltTear1                                                        // Belt tear switch 1 is ok
	            THEN
	                #sUDT_HMIStatus.Specific.BeltTear1Err := FALSE;                // reset error
	            END_IF;

	            // Belt tear switch 2
	            IF #ix_BeltTear2                                                        // Belt tear switch 2 is ok
	            THEN
	                #sUDT_HMIStatus.Specific.BeltTear2Err := FALSE;                // reset error
	            END_IF;

	            // Maintenace supports for lift carriage extracted
	            IF #ix_MaintSupport1                                                    // Maintenace support 1 stowed
	            THEN
	                #sUDT_HMIStatus.Specific.MaintSupport1Err := FALSE;             // reset error
	            END_IF;

	            // Maintenace supports for lift carriage extracted
	            IF #ix_MaintSupport2                                                    // Maintenace support 2 stowed
	            THEN
	                #sUDT_HMIStatus.Specific.MaintSupport2Err := FALSE;             // reset error
	            END_IF;

	            // Upper limit switch
	            IF NOT #ix_LimitSwitchUp                                                // Upper limit switch not overrun
	            THEN
	                #sUDT_HMIStatus.Specific.UpperPositionErr := FALSE;             // reset error
	            END_IF;

	            IF #ix_SafetyDoorDiagUp                                                // Safety door diagnostic output
	            THEN
	                #sUDT_HMIStatus.Specific.SafetyDoorUpErr := FALSE;                 // reset error
	            END_IF;

	            // Lower limit switch
	            IF NOT #ix_LimitSwitchDown                                                // Lower limit switch not overrun
	            THEN
	                #sUDT_HMIStatus.Specific.LowerPositionErr := FALSE;             // reset error
	            END_IF;

	            IF #ix_SafetyDoorDiagDown                                                // Safety door diagnostic output
	            THEN
	                #sUDT_HMIStatus.Specific.SafetyDoorDownErr := FALSE;                 // reset error
	            END_IF;

